(* IEC 61131-3 sources: OpenPLC_Sample_Programs/successed_ST (part 11) *)

        Pusher_states_t#Wait_Metal:
            Pusher2_transit := FALSE;
            Pusher_Timer3_IN := TRUE;
            Pusher_Timer3_PT := Pusher_Duration3;
            IF Pusher_Timer3_IN THEN
                Pusher_Timer3_Q := (Pusher_Timer3_ET = USINT#0);
                IF (Pusher_Timer3_ET > USINT#0) THEN
                    Pusher_Timer3_ET := (Pusher_Timer3_ET - USINT#1);
                ELSE
                    Pusher_Timer3_ET := USINT#0;
                END_IF;
            ELSE
                Pusher_Timer3_Q := FALSE;
                Pusher_Timer3_ET := Pusher_Timer3_PT;
            END_IF;
            Pusher_interconnect3 := Pusher_Timer3_Q;
            IF Pusher_interconnect3 THEN
                Pusher2_transit := TRUE;
                Pusher2_state := Pusher_states_t#Reset_interconnect_Slide3_Metal;
            END_IF;

        Pusher_states_t#Wait_White:
            Pusher2_transit := FALSE;
            Pusher_Timer3_IN := TRUE;
            Pusher_Timer3_PT := Pusher_Duration3;
            IF Pusher_Timer3_IN THEN
                Pusher_Timer3_Q := (Pusher_Timer3_ET = USINT#0);
                IF (Pusher_Timer3_ET > USINT#0) THEN
                    Pusher_Timer3_ET := (Pusher_Timer3_ET - USINT#1);
                ELSE
                    Pusher_Timer3_ET := USINT#0;
                END_IF;
            ELSE
                Pusher_Timer3_Q := FALSE;
                Pusher_Timer3_ET := Pusher_Timer3_PT;
            END_IF;
            Pusher_interconnect3 := Pusher_Timer3_Q;
            IF Pusher_interconnect3 THEN
                Pusher2_transit := TRUE;
                Pusher2_state := Pusher_states_t#Reset_interconnect_Slide3_White;
            END_IF;

        Pusher_states_t#Wait_Y1_Black:
            Pusher2_transit := FALSE;
            IF (Pusher_PusherY1 = TRUE) THEN
                Pusher_Timer3_IN := Pusher_PusherY1;
                Pusher_Timer3_PT := Pusher_Duration3;
                IF Pusher_Timer3_IN THEN
                    Pusher_Timer3_Q := (Pusher_Timer3_ET = USINT#0);
                    IF (Pusher_Timer3_ET > USINT#0) THEN
                        Pusher_Timer3_ET := (Pusher_Timer3_ET - USINT#1);
                    ELSE
                        Pusher_Timer3_ET := USINT#0;
                    END_IF;
                ELSE
                    Pusher_Timer3_Q := FALSE;
                    Pusher_Timer3_ET := Pusher_Timer3_PT;
                END_IF;
                Pusher_interconnect3 := Pusher_Timer3_Q;
            END_IF;
            IF Pusher_interconnect3 THEN
                Pusher2_transit := TRUE;
                Pusher2_state := Pusher_states_t#PusherY1_Move_In_Black;
            END_IF;

        Pusher_states_t#Wait_Y1_Metal:
            Pusher2_transit := FALSE;
            IF (Pusher_PusherY1 = TRUE) THEN
                Pusher_Timer3_IN := Pusher_PusherY1;
                Pusher_Timer3_PT := Pusher_Duration3;
                IF Pusher_Timer3_IN THEN
                    Pusher_Timer3_Q := (Pusher_Timer3_ET = USINT#0);
                    IF (Pusher_Timer3_ET > USINT#0) THEN
                        Pusher_Timer3_ET := (Pusher_Timer3_ET - USINT#1);
                    ELSE
                        Pusher_Timer3_ET := USINT#0;
                    END_IF;
                ELSE
                    Pusher_Timer3_Q := FALSE;
                    Pusher_Timer3_ET := Pusher_Timer3_PT;
                END_IF;
                Pusher_interconnect3 := Pusher_Timer3_Q;
            END_IF;
            IF Pusher_interconnect3 THEN
                Pusher2_transit := TRUE;
                Pusher2_state := Pusher_states_t#PusherY1_Move_In_Metal;
            END_IF;

        Pusher_states_t#Wait_Y1_White:
            Pusher2_transit := FALSE;
            IF (Pusher_PusherY1 = TRUE) THEN
                Pusher_Timer3_IN := Pusher_PusherY1;
                Pusher_Timer3_PT := Pusher_Duration3;
                IF Pusher_Timer3_IN THEN
                    Pusher_Timer3_Q := (Pusher_Timer3_ET = USINT#0);
                    IF (Pusher_Timer3_ET > USINT#0) THEN
                        Pusher_Timer3_ET := (Pusher_Timer3_ET - USINT#1);
                    ELSE
                        Pusher_Timer3_ET := USINT#0;
                    END_IF;
                ELSE
                    Pusher_Timer3_Q := FALSE;
                    Pusher_Timer3_ET := Pusher_Timer3_PT;
                END_IF;
                Pusher_interconnect3 := Pusher_Timer3_Q;
            END_IF;
            IF Pusher_interconnect3 THEN
                Pusher2_transit := TRUE;
                Pusher2_state := Pusher_states_t#PusherY1_Move_In_White;
            END_IF;

        Pusher_states_t#Wait_Y2_Black:
            Pusher2_transit := FALSE;
            IF (Pusher_PusherY2 = TRUE) THEN
                Pusher_Timer3_IN := Pusher_PusherY2;
                Pusher_Timer3_PT := Pusher_Duration3;
                IF Pusher_Timer3_IN THEN
                    Pusher_Timer3_Q := (Pusher_Timer3_ET = USINT#0);
                    IF (Pusher_Timer3_ET > USINT#0) THEN
                        Pusher_Timer3_ET := (Pusher_Timer3_ET - USINT#1);
                    ELSE
                        Pusher_Timer3_ET := USINT#0;
                    END_IF;
                ELSE
                    Pusher_Timer3_Q := FALSE;
                    Pusher_Timer3_ET := Pusher_Timer3_PT;
                END_IF;
                Pusher_interconnect3 := Pusher_Timer3_Q;
            END_IF;
            IF Pusher_interconnect3 THEN
                Pusher2_transit := TRUE;
                Pusher2_state := Pusher_states_t#PusherY2_Move_In_Black;
            END_IF;

        Pusher_states_t#Wait_Y2_Metal:
            Pusher2_transit := FALSE;
            IF (Pusher_PusherY2 = TRUE) THEN
                Pusher_Timer3_IN := Pusher_PusherY2;
                Pusher_Timer3_PT := Pusher_Duration3;
                IF Pusher_Timer3_IN THEN
                    Pusher_Timer3_Q := (Pusher_Timer3_ET = USINT#0);
                    IF (Pusher_Timer3_ET > USINT#0) THEN
                        Pusher_Timer3_ET := (Pusher_Timer3_ET - USINT#1);
                    ELSE
                        Pusher_Timer3_ET := USINT#0;
                    END_IF;
                ELSE
                    Pusher_Timer3_Q := FALSE;
                    Pusher_Timer3_ET := Pusher_Timer3_PT;
                END_IF;
                Pusher_interconnect3 := Pusher_Timer3_Q;
            END_IF;
            IF Pusher_interconnect3 THEN
                Pusher2_transit := TRUE;
                Pusher2_state := Pusher_states_t#PusherY2_Move_In_Metal;
            END_IF;

        Pusher_states_t#Wait_Y2_White:
            Pusher2_transit := FALSE;
            IF (Pusher_PusherY2 = TRUE) THEN
                Pusher_Timer3_IN := Pusher_PusherY2;
                Pusher_Timer3_PT := Pusher_Duration3;
                IF Pusher_Timer3_IN THEN
                    Pusher_Timer3_Q := (Pusher_Timer3_ET = USINT#0);
                    IF (Pusher_Timer3_ET > USINT#0) THEN
                        Pusher_Timer3_ET := (Pusher_Timer3_ET - USINT#1);
                    ELSE
                        Pusher_Timer3_ET := USINT#0;
                    END_IF;
                ELSE
                    Pusher_Timer3_Q := FALSE;
                    Pusher_Timer3_ET := Pusher_Timer3_PT;
                END_IF;
                Pusher_interconnect3 := Pusher_Timer3_Q;
            END_IF;
            IF Pusher_interconnect3 THEN
                Pusher2_transit := TRUE;
                Pusher2_state := Pusher_states_t#PusherY2_Move_In_White;
            END_IF;

            END_CASE;
    IF ((Actuator_SorterGreenLampConveyor AND Actuator_MagazinGreenLamp) AND Actuator_StampGreenLamp) THEN
        IF (((Stamp_StartCommandStamp AND Crane_StartCommandCrane) AND Conveyor_StartCommandConveyor) AND Mag_StartCommandMagazin) THEN
            Crane_StartVar := TRUE;
            Conveyor_StartVar := TRUE;
            Mag_StartVar := TRUE;
            Pusher_StartVar := TRUE;
            Stamp_StartVar := TRUE;
            DIAGNOSIS_ACTIVE := TRUE;
        END_IF;
    END_IF;
    Crane_SFCReset := FALSE;
    Conveyor_SFCReset := FALSE;
    Mag_SFCReset := FALSE;
    Pusher_SFCReset := FALSE;
    Stamp_SFCReset := FALSE;

    Crane_AnalogCranePressure := PARAMETER_CRANE_PRESSURE_METALLIC;

ELSIF ((NOT Sensor_SorterEmergencyStop OR NOT Sensor_StampEmergencyStop) OR NOT Sensor_MagazinEmergencyStop) THEN
    Actuator_MagazinSlider := FALSE;
    Actuator_CraneLower := FALSE;
    Actuator_MagazinVacuumOn := FALSE;
    Actuator_MagazinVacuumOff := TRUE;
    Actuator_MagazinGreenLamp := FALSE;
    Actuator_CraneTurnCounterclockwise := FALSE;
    Actuator_CraneTurnClockwise := FALSE;
    Actuator_SorterConveyorTowardsStacker := FALSE;
    Actuator_SorterConveyorTowardsCrane := FALSE;
    Actuator_SorterGreenLampConveyor := FALSE;
    Actuator_PusherY1 := FALSE;
    Actuator_PusherY2 := FALSE;
    Actuator_StampSliderMovedOut := TRUE;
    Actuator_StampSliderMovedIn := FALSE;
    Actuator_StampGreenLamp := FALSE;
    Actuator_StampPusher := FALSE;
    Actuator_AnalogCranePressure := 0;
    Crane_SFCReset := TRUE;
    Conveyor_SFCReset := TRUE;
    Mag_SFCReset := TRUE;
    Pusher_SFCReset := TRUE;
    Stamp_SFCReset := TRUE;
    Crane_StartVar := FALSE;
    Conveyor_StartVar := FALSE;
    Mag_StartVar := FALSE;
    Pusher_StartVar := FALSE;
    Stamp_StartVar := FALSE;
END_IF;

END_PROGRAM

CONFIGURATION Config0
  RESOURCE Res0 ON PLC
    TASK task0(INTERVAL := T#50ms, PRIORITY := 0);
    PROGRAM instance0 WITH task0 : Main;
  END_RESOURCE
END_CONFIGURATION

(* ---- Code_3.st ---- *)
TYPE
Crane3_states_t : (Crane_Init,Crane_Go_Up , Crane_Init_2 , Crane_Lift_At_Stamp
, Crane_Lift_Conveyor , Crane_Lift_Magazin , Crane_Lift_Magazin_Metallic ,
Crane_Lower , Crane_On_Conveyor , Crane_On_Conveyor_Metallic ,
Crane_On_Stamp_Metallic , Crane_Turn_Left_From_Stamp , Crane_Turn_Left_Metallic
, Crane_Turn_Left_NOT_Metallic , Init , Interstep , Interstep_2 ,
Interstep_Check_Workpiece , Lower_Crane , Reset_interconnect , Start_Crane ,
Step0 , Step2 , Suck_At_Stamp , TimeDelay , Turn_Right , Wait_At_Stamp , pause ,
release , release_Workpiece);
END_TYPE

PROGRAM Crane3
    VAR  Duration1 : TIME := T#1s500ms; END_VAR
    VAR  SFCInit : BOOL; END_VAR
    VAR  TimeDelay_Timer : TON; END_VAR
    VAR  TimeDelay_Timer_Duration : TIME := T#50ms; END_VAR
    VAR  TimeDelay_Timer_interconnect : BOOL; END_VAR
    VAR  Timer1 : TON; END_VAR
    VAR  _state : Crane3_states_t; END_VAR
    VAR  _transit : BOOL; END_VAR
    VAR  actualtime1 : TIME; END_VAR
    VAR  interconnect : BOOL; END_VAR
    VAR  interconnectCraneStartCommand : BOOL; END_VAR

    VAR_INPUT  CraneDown : BOOL; END_VAR
    VAR_INPUT  CraneOnConveyor : BOOL; END_VAR
    VAR_INPUT  CraneOnMagazin : BOOL; END_VAR
    VAR_INPUT  CranePositionStamp : BOOL; END_VAR
    VAR_INPUT  CraneSucked : BOOL; END_VAR
    VAR_INPUT  CraneUp : BOOL; END_VAR
    VAR_INPUT  MagazinCapacitiveSensor : BOOL; END_VAR
    VAR_INPUT  SFCReset : BOOL; END_VAR
    VAR_INPUT  SliderMovedOut : BOOL; END_VAR
    VAR_INPUT  SliderNotMovedOut : BOOL; END_VAR
    VAR_INPUT  StampLowered : BOOL; END_VAR
    VAR_INPUT  StampSliderFilled : BOOL; END_VAR
    VAR_INPUT  StartButtonMagazin : BOOL; END_VAR
    VAR_INPUT  StartVar : BOOL; END_VAR
    VAR_INPUT  WorkpieceReady : BOOL; END_VAR

    VAR_OUTPUT  CraneLower : BOOL; END_VAR
    VAR_OUTPUT  CraneTurnClockwise : BOOL; END_VAR
    VAR_OUTPUT  CraneTurnCounterclockwise : BOOL; END_VAR
    VAR_OUTPUT  MagazinVacuumOff : BOOL; END_VAR
    VAR_OUTPUT  MagazinVacuumOn : BOOL; END_VAR
    VAR_OUTPUT  StartCommandCrane : BOOL; END_VAR

    CASE _state OF
        Crane3_states_t#Crane_Go_Up:
            _transit := FALSE;
            CraneLower := FALSE;
            IF CraneUp THEN
                _transit := TRUE;
                _state := Crane3_states_t#pause;
            END_IF;
        Crane3_states_t#Crane_Init:
            _transit := FALSE;
            CraneLower := TRUE;
            interconnectCraneStartCommand := FALSE;
            IF CraneDown THEN
                _transit := TRUE;
                _state := Crane3_states_t#Crane_Init_2;
            END_IF;
        Crane3_states_t#Crane_Init_2:
            _transit := FALSE;
            CraneLower := FALSE;
            IF CraneUp THEN
                _transit := TRUE;
                _state := Crane3_states_t#Interstep;
            END_IF;
        Crane3_states_t#Crane_Lift_At_Stamp:
            _transit := FALSE;
            CraneLower := FALSE;
            IF CraneUp THEN
                _transit := TRUE;
                _state := Crane3_states_t#Crane_Turn_Left_From_Stamp;
            END_IF;
        Crane3_states_t#Crane_Lift_Conveyor:
            _transit := FALSE;
            CraneLower := FALSE;
            IF TRUE THEN
                _transit := TRUE;
                _state := Crane3_states_t#Interstep;
            END_IF;
        Crane3_states_t#Crane_Lift_Magazin:
            _transit := FALSE;
            CraneLower := FALSE;
            IF CraneUp THEN
                _transit := TRUE;
                _state := Crane3_states_t#Crane_Turn_Left_NOT_Metallic;
            END_IF;
        Crane3_states_t#Crane_Lift_Magazin_Metallic:
            _transit := FALSE;
            CraneLower := FALSE;
            IF CraneUp THEN
                _transit := TRUE;
                _state := Crane3_states_t#Crane_Turn_Left_Metallic;
            END_IF;
        Crane3_states_t#Crane_Lower:
            _transit := FALSE;
            MagazinVacuumOn := TRUE;
            MagazinVacuumOff := FALSE;
            CraneLower := TRUE;
            IF CraneSucked THEN
                _transit := TRUE;
                _state := Crane3_states_t#Step0;
            END_IF;
        Crane3_states_t#Crane_On_Conveyor:
            _transit := FALSE;
            CraneTurnCounterclockwise := FALSE;
            CraneTurnClockwise := FALSE;
            CraneLower := TRUE;
            IF CraneDown THEN
                _transit := TRUE;
                _state := Crane3_states_t#release;
            END_IF;
        Crane3_states_t#Crane_On_Conveyor_Metallic:
            _transit := FALSE;
            CraneTurnCounterclockwise := FALSE;
            CraneTurnClockwise := FALSE;
            CraneLower := TRUE;
            IF CraneDown THEN
                _transit := TRUE;
                _state := Crane3_states_t#release;
            END_IF;
        Crane3_states_t#Crane_On_Stamp_Metallic:
            _transit := FALSE;
            CraneTurnCounterclockwise := FALSE;
            CraneTurnClockwise := FALSE;
            CraneLower := TRUE;
            IF CraneDown THEN
                _transit := TRUE;
                _state := Crane3_states_t#release_Workpiece;
            END_IF;
        Crane3_states_t#Crane_Turn_Left_From_Stamp:
            _transit := FALSE;
            CraneTurnClockwise := TRUE;
            CraneTurnCounterclockwise := FALSE;
            IF CraneOnConveyor THEN
                _transit := TRUE;
                _state := Crane3_states_t#Crane_On_Conveyor_Metallic;
            END_IF;
        Crane3_states_t#Crane_Turn_Left_Metallic:
            _transit := FALSE;
            CraneTurnCounterclockwise := TRUE;
            CraneTurnClockwise := FALSE;
            IF CranePositionStamp THEN
                _transit := TRUE;
                _state := Crane3_states_t#Crane_On_Stamp_Metallic;
            END_IF;
        Crane3_states_t#Crane_Turn_Left_NOT_Metallic:
            _transit := FALSE;
            CraneTurnCounterclockwise := TRUE;
            CraneTurnClockwise := FALSE;
            IF CraneOnConveyor THEN
                _transit := TRUE;
                _state := Crane3_states_t#Crane_On_Conveyor;
            END_IF;
        Crane3_states_t#Init:
            _transit := FALSE;
            IF TRUE THEN
                _transit := TRUE;
                _state := Crane3_states_t#Start_Crane;
            END_IF;
        Crane3_states_t#Interstep:
            _transit := FALSE;
            StartCommandCrane := TRUE;
            IF StartVar THEN
                _transit := TRUE;
                _state := Crane3_states_t#Interstep_2;
            END_IF;
        Crane3_states_t#Interstep_2:
            _transit := FALSE;
            IF SliderMovedOut THEN
                _transit := TRUE;
                _state := Crane3_states_t#TimeDelay;
            END_IF;
        Crane3_states_t#Interstep_Check_Workpiece:
            _transit := FALSE;
            CraneTurnClockwise := FALSE;
            CraneTurnCounterclockwise := FALSE;
            IF (NOT WorkpieceReady AND StampSliderFilled) THEN
                _transit := TRUE;
                _state := Crane3_states_t#Wait_At_Stamp;
            ELSIF (NOT WorkpieceReady AND NOT StampSliderFilled) THEN
                _transit := TRUE;
                _state := Crane3_states_t#Step2;
            ELSIF WorkpieceReady THEN
                _transit := TRUE;
                _state := Crane3_states_t#Crane_Lower;
            END_IF;
        Crane3_states_t#Lower_Crane:
            _transit := FALSE;
            CraneLower := TRUE;
            IF CraneDown THEN
                _transit := TRUE;
                _state := Crane3_states_t#Suck_At_Stamp;
            END_IF;
        Crane3_states_t#Reset_interconnect:
            _transit := FALSE;
            interconnect := FALSE;
            Timer1(IN := FALSE, PT := TIME#1ms);
            IF SliderMovedOut THEN
                _transit := TRUE;
                _state := Crane3_states_t#Lower_Crane;
            END_IF;
        Crane3_states_t#Start_Crane:
            _transit := FALSE;
            CraneLower := FALSE;
            MagazinVacuumOff := TRUE;
            MagazinVacuumOn := FALSE;
            CraneTurnCounterclockwise := FALSE;
            CraneTurnClockwise := FALSE;
            StartVar := FALSE;
            StartCommandCrane := FALSE;
            IF (StartButtonMagazin = TRUE) THEN
                interconnectCraneStartCommand := TRUE;
            END_IF;
            IF interconnectCraneStartCommand THEN
                _transit := TRUE;
                _state := Crane3_states_t#Crane_Init;
            END_IF;
        Crane3_states_t#Step0:
            _transit := FALSE;
            IF NOT MagazinCapacitiveSensor THEN
                _transit := TRUE;
                _state := Crane3_states_t#Crane_Lift_Magazin;
            ELSIF MagazinCapacitiveSensor THEN
                _transit := TRUE;
                _state := Crane3_states_t#Crane_Lift_Magazin_Metallic;
            END_IF;
        Crane3_states_t#Step2:
            _transit := FALSE;
            IF TRUE THEN
                _transit := TRUE;
                _state := Crane3_states_t#Start_Crane;
            END_IF;
        Crane3_states_t#Suck_At_Stamp:
            _transit := FALSE;
            MagazinVacuumOn := TRUE;
            MagazinVacuumOff := FALSE;
            IF CraneSucked THEN
                _transit := TRUE;
                _state := Crane3_states_t#Crane_Lift_At_Stamp;
            END_IF;
        Crane3_states_t#TimeDelay:
            _transit := FALSE;
            TimeDelay_Timer(IN := TRUE, PT := TimeDelay_Timer_Duration);
            TimeDelay_Timer_interconnect := TimeDelay_Timer.Q;
            IF TimeDelay_Timer_interconnect THEN
                _transit := TRUE;
                _state := Crane3_states_t#Turn_Right;
            END_IF;
        Crane3_states_t#Turn_Right:
             _transit := FALSE;
             CraneTurnClockwise := TRUE;
             CraneTurnCounterclockwise := FALSE;
             IF CraneOnMagazin THEN
                _transit := TRUE;
                _state := Crane3_states_t#Interstep_Check_Workpiece;
             END_IF;
        Crane3_states_t#Wait_At_Stamp:
            _transit := FALSE;
            IF TRUE THEN
                _transit := TRUE;
                _state := Crane3_states_t#pause;
            END_IF;
        Crane3_states_t#pause:
            _transit := FALSE;
            Timer1(IN := CraneUp, PT := Duration1);
            interconnect := Timer1.Q;
            IF interconnect THEN
                _transit := TRUE;
                _state := Crane3_states_t#Reset_interconnect;
            END_IF;
        Crane3_states_t#release:
            _transit := FALSE;
            MagazinVacuumOff := TRUE;
            MagazinVacuumOn := FALSE;
            IF TRUE THEN
                _transit := TRUE;
                _state := Crane3_states_t#Crane_Lift_Conveyor;
            END_IF;
        Crane3_states_t#release_Workpiece:
            _transit := FALSE;
            MagazinVacuumOff := TRUE;
            MagazinVacuumOn := FALSE;
            IF TRUE THEN
                _transit := TRUE;
                _state := Crane3_states_t#Crane_Go_Up;
            END_IF;
        END_CASE;
END_PROGRAM

CONFIGURATION Config0
  RESOURCE Res0 ON PLC
    TASK task0(INTERVAL := T#50ms, PRIORITY := 0);
    PROGRAM instance0 WITH task0 : Crane3;
  END_RESOURCE
END_CONFIGURATION

(* ---- Code_5.st ---- *)
TYPE
Crane5_states_t : (Crane_Init ,Crane_Go_Up ,  Crane_Init_2 , Crane_Lift_At_Stamp
, Crane_Lift_Conveyor , Crane_Lift_Conveyor_Black , Crane_Lift_Magazin ,
Crane_Lift_Magazin_Metallic , Crane_Lift_NOT_Metallic_Black , Crane_Lower ,
Crane_On_Conveyor , Crane_On_Conveyor_Metallic ,
Crane_On_Conveyor_Not_Metallica_Black , Crane_On_Stamp_Metallic ,
Crane_On_Stamp_Stop_Black , Crane_Turn_Left_Back_To_Stamp ,
Crane_Turn_Left_From_Stamp , Crane_Turn_Left_Metallic ,
Crane_Turn_Left_NOT_Metallic , Crane_Turn_Left_NOT_Metallic_Black , Init ,
Interstep , Interstep_2 , Last_Workpiece_At_Stamp , Lower_Crane , Magazin_Stop ,
Magazin_Stop_Black , No_Workpiece_ready , Reset_interconnect , Start_Crane ,
Step0 , Suck_At_Stamp , TimeDelay , Turn_Right , Turn_Right_Black , pause ,
release , release_Black , release_Workpiece);
END_TYPE

PROGRAM Crane5
    VAR  CranTurnClockwise : BOOL; END_VAR
    VAR_INPUT  CraneDown : BOOL; END_VAR
    VAR_OUTPUT  CraneLower : BOOL; END_VAR
    VAR_INPUT  CraneOnConveyor : BOOL; END_VAR
    VAR_INPUT  CraneOnMagazin : BOOL; END_VAR
    VAR_INPUT  CranePositionStamp : BOOL; END_VAR
    VAR_INPUT  CraneSucked : BOOL; END_VAR
    VAR_OUTPUT  CraneTurnClockwise : BOOL; END_VAR
    VAR_OUTPUT  CraneTurnCounterclockwise : BOOL; END_VAR
    VAR_INPUT  CraneUp : BOOL; END_VAR
    VAR  Duration1 : TIME := TIME#1s500ms; END_VAR
    VAR_INPUT  MagazinCapacitiveSensor : BOOL; END_VAR
    VAR_OUTPUT  MagazinVacuumOff : BOOL; END_VAR
    VAR_OUTPUT  MagazinVacuumOn : BOOL; END_VAR
    VAR  SFCInit : BOOL; END_VAR
    VAR_INPUT  SFCReset : BOOL; END_VAR
    VAR_INPUT  SliderMovedOut : BOOL; END_VAR
    VAR_INPUT  SliderNotMovedOut : BOOL; END_VAR
    VAR_INPUT  StampLowered : BOOL; END_VAR
    VAR_INPUT  StampSliderFilled : BOOL; END_VAR
    VAR_INPUT  StartButtonMagazin : BOOL; END_VAR
    VAR_OUTPUT  StartCommandCrane : BOOL; END_VAR
    VAR_INPUT  StartVar : BOOL; END_VAR
    VAR  TimeDelay_Timer : TON; END_VAR
    VAR  TimeDelay_Timer_Duration : TIME := TIME#50.0ms; END_VAR
    VAR  TimeDelay_Timer_interconnect : BOOL; END_VAR
    VAR  Timer1 : TON; END_VAR
    VAR_INPUT  WorkpieceReady : BOOL; END_VAR
    VAR  _state : Crane5_states_t; END_VAR
    VAR  _transit : BOOL; END_VAR
    VAR  actualtime1 : TIME; END_VAR
    VAR  interconnect : BOOL; END_VAR
    VAR  interconnectCraneStartCommand : BOOL; END_VAR

    CASE _state OF
        Crane5_states_t#Crane_Go_Up:
            _transit := FALSE;
            CraneLower := FALSE;
            IF (CraneUp AND (MagazinCapacitiveSensor OR NOT WorkpieceReady)) THEN
                _transit := TRUE;
                _state := Crane5_states_t#pause;
            ELSIF ((CraneUp AND NOT MagazinCapacitiveSensor) AND WorkpieceReady) THEN
                _transit := TRUE;
                _state := Crane5_states_t#Turn_Right_Black;
            END_IF;
        Crane5_states_t#Crane_Init:
            _transit := FALSE;
            CraneLower := TRUE;
            interconnectCraneStartCommand := FALSE;
            IF CraneDown THEN
                _transit := TRUE;
                _state := Crane5_states_t#Crane_Init_2;
            END_IF;
        Crane5_states_t#Crane_Init_2:
            _transit := FALSE;
            CraneLower := FALSE;
            IF CraneUp THEN
                _transit := TRUE;
                _state := Crane5_states_t#Interstep;
            END_IF;
        Crane5_states_t#Crane_Lift_At_Stamp:
            _transit := FALSE;
            CraneLower := FALSE;
            IF CraneUp THEN
                _transit := TRUE;
                _state := Crane5_states_t#Crane_Turn_Left_From_Stamp;
            END_IF;
        Crane5_states_t#Crane_Lift_Conveyor:
            _transit := FALSE;
            CraneLower := FALSE;
            IF TRUE THEN
                _transit := TRUE;
                _state := Crane5_states_t#Interstep;
            END_IF;
        Crane5_states_t#Crane_Lift_Conveyor_Black:
            _transit := FALSE;
            CraneLower := FALSE;
            IF CraneUp THEN
                _transit := TRUE;
                _state := Crane5_states_t#Crane_Turn_Left_Back_To_Stamp;
            END_IF;
        Crane5_states_t#Crane_Lift_Magazin:
            _transit := FALSE;
            CraneLower := FALSE;
            IF CraneUp THEN
                _transit := TRUE;
                _state := Crane5_states_t#Crane_Turn_Left_NOT_Metallic;
            END_IF;
        Crane5_states_t#Crane_Lift_Magazin_Metallic:
            _transit := FALSE;
            CraneLower := FALSE;
            IF CraneUp THEN
                _transit := TRUE;
                _state := Crane5_states_t#Crane_Turn_Left_Metallic;
            END_IF;
        Crane5_states_t#Crane_Lift_NOT_Metallic_Black:
            _transit := FALSE;
            CraneLower := FALSE;
            IF CraneUp THEN
                _transit := TRUE;
                _state := Crane5_states_t#Crane_Turn_Left_NOT_Metallic_Black;
            END_IF;
        Crane5_states_t#Crane_Lower:
            _transit := FALSE;
            MagazinVacuumOn := TRUE;
            MagazinVacuumOff := FALSE;
            CraneLower := TRUE;
            IF CraneSucked THEN
                _transit := TRUE;
                _state := Crane5_states_t#Step0;
            END_IF;
        Crane5_states_t#Crane_On_Conveyor:
            _transit := FALSE;
            CraneTurnCounterclockwise := FALSE;
            CraneTurnClockwise := FALSE;
            CraneLower := TRUE;
            IF CraneDown THEN
                _transit := TRUE;
                _state := Crane5_states_t#release;
            END_IF;
        Crane5_states_t#Crane_On_Conveyor_Metallic:
            _transit := FALSE;
            CraneTurnCounterclockwise := FALSE;
            CraneTurnClockwise := FALSE;
            CraneLower := TRUE;
            IF CraneDown THEN
                _transit := TRUE;
                _state := Crane5_states_t#release;
            END_IF;
        Crane5_states_t#Crane_On_Conveyor_Not_Metallica_Black:
            _transit := FALSE;
            CraneTurnCounterclockwise := FALSE;
            CraneTurnClockwise := FALSE;
            CraneLower := TRUE;
            IF CraneDown THEN
                _transit := TRUE;
                _state := Crane5_states_t#release_Black;
            END_IF;
        Crane5_states_t#Crane_On_Stamp_Metallic:
            _transit := FALSE;
            CraneTurnCounterclockwise := FALSE;
            CraneTurnClockwise := FALSE;
            CraneLower := TRUE;
            IF CraneDown THEN
                _transit := TRUE;
                _state := Crane5_states_t#release_Workpiece;
            END_IF;
        Crane5_states_t#Crane_On_Stamp_Stop_Black:
            _transit := FALSE;
            CraneTurnClockwise := FALSE;
            CraneTurnCounterclockwise := FALSE;
            IF TRUE THEN
                _transit := TRUE;
                _state := Crane5_states_t#Reset_interconnect;
            END_IF;
        Crane5_states_t#Crane_Turn_Left_Back_To_Stamp:
            _transit := FALSE;
            CraneTurnCounterclockwise := TRUE;
            CraneTurnClockwise := FALSE;
            IF CranePositionStamp THEN
                _transit := TRUE;
                _state := Crane5_states_t#Crane_On_Stamp_Stop_Black;
            END_IF;
        Crane5_states_t#Crane_Turn_Left_From_Stamp:
            _transit := FALSE;
            CraneTurnClockwise := TRUE;
            CraneTurnCounterclockwise := FALSE;
            IF CraneOnConveyor THEN
                _transit := TRUE;
                _state := Crane5_states_t#Crane_On_Conveyor_Metallic;
            END_IF;
        Crane5_states_t#Crane_Turn_Left_Metallic:
            _transit := FALSE;
            CraneTurnCounterclockwise := TRUE;
            CraneTurnClockwise := FALSE;
            IF CranePositionStamp THEN
                _transit := TRUE;
                _state := Crane5_states_t#Crane_On_Stamp_Metallic;
            END_IF;
        Crane5_states_t#Crane_Turn_Left_NOT_Metallic:
            _transit := FALSE;
            CraneTurnCounterclockwise := TRUE;
            CraneTurnClockwise := FALSE;
            IF CraneOnConveyor THEN
                _transit := TRUE;
                _state := Crane5_states_t#Crane_On_Conveyor;
            END_IF;
        Crane5_states_t#Crane_Turn_Left_NOT_Metallic_Black:
            _transit := FALSE;
            CraneTurnCounterclockwise := TRUE;
            CraneTurnClockwise := FALSE;
            IF CraneOnConveyor THEN
                _transit := TRUE;
                _state := Crane5_states_t#Crane_On_Conveyor_Not_Metallica_Black;
            END_IF;
        Crane5_states_t#Init:
            _transit := FALSE;
            IF TRUE THEN
                _transit := TRUE;
                _state := Crane5_states_t#Start_Crane;
            END_IF;
        Crane5_states_t#Interstep:
            _transit := FALSE;
            StartCommandCrane := TRUE;
            IF StartVar THEN
                _transit := TRUE;
                _state := Crane5_states_t#Interstep_2;
            END_IF;
        Crane5_states_t#Interstep_2:
            _transit := FALSE;
            IF SliderMovedOut THEN
                _transit := TRUE;
                _state := Crane5_states_t#TimeDelay;
            END_IF;
        Crane5_states_t#Last_Workpiece_At_Stamp:
            _transit := FALSE;
            IF TRUE THEN
                _transit := TRUE;
                _state := Crane5_states_t#pause;
            END_IF;
        Crane5_states_t#Lower_Crane:
            _transit := FALSE;
            CraneLower := TRUE;
            IF CraneDown THEN
                _transit := TRUE;
                _state := Crane5_states_t#Suck_At_Stamp;
            END_IF;
        Crane5_states_t#Magazin_Stop:
            _transit := FALSE;
            CraneTurnClockwise := FALSE;
            CraneTurnCounterclockwise := FALSE;
            IF WorkpieceReady THEN
                _transit := TRUE;
                _state := Crane5_states_t#Crane_Lower;
            ELSIF (NOT WorkpieceReady AND NOT StampSliderFilled) THEN
                _transit := TRUE;
                _state := Crane5_states_t#No_Workpiece_ready;
            ELSIF (NOT WorkpieceReady AND StampSliderFilled) THEN
                _transit := TRUE;
                _state := Crane5_states_t#Last_Workpiece_At_Stamp;
            END_IF;
        Crane5_states_t#Magazin_Stop_Black:
            _transit := FALSE;
            CraneTurnClockwise := FALSE;
            CraneTurnCounterclockwise := FALSE;
            MagazinVacuumOn := TRUE;
            MagazinVacuumOff := FALSE;
            CraneLower := TRUE;
            IF CraneSucked THEN
                _transit := TRUE;
                _state := Crane5_states_t#Crane_Lift_NOT_Metallic_Black;
            END_IF;
        Crane5_states_t#No_Workpiece_ready:
            _transit := FALSE;
            IF TRUE THEN
                _transit := TRUE;
                _state := Crane5_states_t#Start_Crane;
            END_IF;
        Crane5_states_t#Reset_interconnect:
            _transit := FALSE;
            interconnect := FALSE;
            Timer1(IN := FALSE, PT := TIME#1.0ms);
            IF SliderMovedOut THEN
                _transit := TRUE;
                _state := Crane5_states_t#Lower_Crane;
            END_IF;
        Crane5_states_t#Start_Crane:
            _transit := FALSE;
            CraneLower := FALSE;
            MagazinVacuumOff := TRUE;
            MagazinVacuumOn := FALSE;
            CraneTurnCounterclockwise := FALSE;
            CraneTurnClockwise := FALSE;
            StartVar := FALSE;
            StartCommandCrane := FALSE;
            IF (StartButtonMagazin = TRUE) THEN
                interconnectCraneStartCommand := TRUE;
            END_IF;
            IF interconnectCraneStartCommand THEN
                _transit := TRUE;
                _state := Crane5_states_t#Crane_Init;
            END_IF;
        Crane5_states_t#Step0:
            _transit := FALSE;
            IF NOT MagazinCapacitiveSensor THEN
                _transit := TRUE;
                _state := Crane5_states_t#Crane_Lift_Magazin;
            ELSIF MagazinCapacitiveSensor THEN
                _transit := TRUE;
                _state := Crane5_states_t#Crane_Lift_Magazin_Metallic;
            END_IF;
        Crane5_states_t#Suck_At_Stamp:
            _transit := FALSE;
            MagazinVacuumOn := TRUE;
            MagazinVacuumOff := FALSE;
            IF CraneSucked THEN
                _transit := TRUE;
                _state := Crane5_states_t#Crane_Lift_At_Stamp;
            END_IF;
        Crane5_states_t#TimeDelay:
            _transit := FALSE;
            TimeDelay_Timer(IN := TRUE, PT := TimeDelay_Timer_Duration);
            TimeDelay_Timer_interconnect := TimeDelay_Timer.Q;
            IF TimeDelay_Timer_interconnect THEN
                _transit := TRUE;
                _state := Crane5_states_t#Turn_Right;
            END_IF;
        Crane5_states_t#Turn_Right:
            _transit := FALSE;
            CraneTurnClockwise := TRUE;
            CraneTurnCounterclockwise := FALSE;
            IF CraneOnMagazin THEN
                _transit := TRUE;
                _state := Crane5_states_t#Magazin_Stop;
            END_IF;
        Crane5_states_t#Turn_Right_Black:
            _transit := FALSE;
            CraneTurnClockwise := TRUE;
            CraneTurnCounterclockwise := FALSE;
            IF CraneOnMagazin THEN
                _transit := TRUE;
                _state := Crane5_states_t#Magazin_Stop_Black;
            END_IF;
        Crane5_states_t#pause:
            _transit := FALSE;
            Timer1(IN := CraneUp, PT := Duration1);
            interconnect := Timer1.Q;
            IF interconnect THEN
                _transit := TRUE;
                _state := Crane5_states_t#Reset_interconnect;
            END_IF;
        Crane5_states_t#release:
            _transit := FALSE;
            MagazinVacuumOff := TRUE;
            MagazinVacuumOn := FALSE;
            IF TRUE THEN
                _transit := TRUE;
                _state := Crane5_states_t#Crane_Lift_Conveyor;
            END_IF;
        Crane5_states_t#release_Black:
            _transit := FALSE;
            MagazinVacuumOn := FALSE;
            MagazinVacuumOff := TRUE;
            IF TRUE THEN
                _transit := TRUE;
                _state := Crane5_states_t#Crane_Lift_Conveyor_Black;
            END_IF;
        Crane5_states_t#release_Workpiece:
            _transit := FALSE;
            MagazinVacuumOff := TRUE;
            MagazinVacuumOn := FALSE;
            IF TRUE THEN
                _transit := TRUE;
                _state := Crane5_states_t#Crane_Go_Up;
            END_IF;
    END_CASE;
END_PROGRAM

CONFIGURATION Config0
  RESOURCE Res0 ON PLC
    TASK task0(INTERVAL := T#50ms, PRIORITY := 0);
    PROGRAM instance0 WITH task0 : Crane5;
  END_RESOURCE
END_CONFIGURATION

(* ---- constantprogram.st ---- *)
PROGRAM CONSTANTPROGRAM
    VAR_INPUT
        I : INT;
    END_VAR

    VAR_OUTPUT
        O : INT;
        C : INT;
    END_VAR

    O := I;
    C := 42;

END_PROGRAM

CONFIGURATION Config0
  RESOURCE Res0 ON PLC
    TASK TASK0(INTERVAL := T#50MS, PRIORITY := 0);
    PROGRAM INSTANCE0 WITH TASK0 : CONSTANTPROGRAM;
  END_RESOURCE
END_CONFIGURATION

(* ---- Crane.st ---- *)
TYPE
    CRANE_STATES_T : (CRANE_GO_UP , CRANE_INIT , CRANE_INIT_2 , CRANE_LIFT_AT_STAMP , CRANE_LIFT_CONVEYOR , CRANE_LIFT_CONVEYOR_BLACK , CRANE_LIFT_MAGAZIN , CRANE_LIFT_MAGAZIN_METALLIC , CRANE_LIFT_NOT_METALLIC_BLACK , CRANE_LOWER , CRANE_ON_CONVEYOR , CRANE_ON_CONVEYOR_METALLIC , CRANE_ON_CONVEYOR_NOT_METALLICA_BLACK , CRANE_ON_STAMP_METALLIC , CRANE_ON_STAMP_STOP_BLACK , CRANE_TURN_LEFT_BACK_TO_STAMP , CRANE_TURN_LEFT_FROM_STAMP , CRANE_TURN_LEFT_METALLIC , CRANE_TURN_LEFT_NOT_METALLIC , CRANE_TURN_LEFT_NOT_METALLIC_BLACK , INIT , INTERSTEP , INTERSTEP_2 , LAST_WORKPIECE_AT_STAMP , LOWER_CRANE , MAGAZIN_STOP , MAGAZIN_STOP_BLACK , NO_WORKPIECE_READY , RESET_INTERCONNECT , START_CRANE , STEP0 , SUCK_AT_STAMP , TIMEDELAY , TURN_RIGHT , TURN_RIGHT_BLACK , PAUSE , RELEASE , RELEASE_BLACK , RELEASE_WORKPIECE);
END_TYPE

PROGRAM CRANE
    VAR  CRANTURNCLOCKWISE : BOOL; END_VAR
    VAR_INPUT  CRANEDOWN : BOOL; END_VAR
    VAR_OUTPUT  CRANELOWER : BOOL; END_VAR
    VAR_INPUT  CRANEONCONVEYOR : BOOL; END_VAR
    VAR_INPUT  CRANEONMAGAZIN : BOOL; END_VAR
    VAR_INPUT  CRANEPOSITIONSTAMP : BOOL; END_VAR
    VAR_INPUT  CRANESUCKED : BOOL; END_VAR
    VAR_OUTPUT  CRANETURNCLOCKWISE : BOOL; END_VAR
    VAR_OUTPUT  CRANETURNCOUNTERCLOCKWISE : BOOL; END_VAR
    VAR_INPUT  CRANEUP : BOOL; END_VAR
    VAR  DURATION1 : TIME := TIME#1S500MS; END_VAR
    VAR_INPUT  MAGAZINCAPACITIVESENSOR : BOOL; END_VAR
    VAR_OUTPUT  MAGAZINSLIDER : BOOL; END_VAR
    VAR_OUTPUT  MAGAZINVACUUMOFF : BOOL; END_VAR
    VAR_OUTPUT  MAGAZINVACUUMON : BOOL; END_VAR
    VAR  SFCINIT : BOOL; END_VAR
    VAR_INPUT  SFCRESET : BOOL; END_VAR
    VAR_INPUT  SLIDERMOVEDOUT : BOOL; END_VAR
    VAR_INPUT  SLIDERNOTMOVEDOUT : BOOL; END_VAR
    VAR_INPUT  STAMPLOWERED : BOOL; END_VAR
    VAR_INPUT  STAMPSLIDERFILLED : BOOL; END_VAR
    VAR_INPUT  STARTBUTTONMAGAZIN : BOOL; END_VAR
    VAR_OUTPUT  STARTCOMMANDCRANE : BOOL; END_VAR
    VAR_INPUT  STARTVAR : BOOL; END_VAR
    VAR  TIMEDELAY_TIMER : TON; END_VAR
    VAR  TIMEDELAY_TIMER_DURATION : TIME := TIME#50MS; END_VAR
    VAR  TIMEDELAY_TIMER_INTERCONNECT : BOOL; END_VAR
    VAR  TIMER1 : TON; END_VAR
    VAR_INPUT  WORKPIECEREADY : BOOL; END_VAR
    VAR  _STATE : CRANE_STATES_T := CRANE_STATES_T#INIT; END_VAR
    VAR  _TRANSIT : BOOL; END_VAR
    VAR  ACTUALTIME1 : TIME; END_VAR
    VAR  INTERCONNECT : BOOL; END_VAR
    VAR  INTERCONNECTCRANESTARTCOMMAND : BOOL; END_VAR

    IF SFCRESET THEN
        _STATE := CRANE_STATES_T#INIT;
    END_IF;

    CASE _STATE OF
        CRANE_STATES_T#CRANE_GO_UP:
            _TRANSIT := FALSE;
            CRANELOWER := FALSE;
            IF (CRANEUP AND (MAGAZINCAPACITIVESENSOR OR NOT WORKPIECEREADY)) THEN
                _TRANSIT := TRUE;
                _STATE := CRANE_STATES_T#PAUSE;
            ELSIF ((CRANEUP AND NOT MAGAZINCAPACITIVESENSOR) AND WORKPIECEREADY) THEN
                _TRANSIT := TRUE;
                _STATE := CRANE_STATES_T#TURN_RIGHT_BLACK;
            END_IF;

        CRANE_STATES_T#CRANE_INIT:
            _TRANSIT := FALSE;
            CRANELOWER := TRUE;
            INTERCONNECTCRANESTARTCOMMAND := FALSE;
            IF CRANEDOWN THEN
                _TRANSIT := TRUE;
                _STATE := CRANE_STATES_T#CRANE_INIT_2;
            END_IF;

        CRANE_STATES_T#CRANE_INIT_2:
            _TRANSIT := FALSE;
            CRANELOWER := FALSE;
            IF CRANEUP THEN
                _TRANSIT := TRUE;
                _STATE := CRANE_STATES_T#INTERSTEP;
            END_IF;

        CRANE_STATES_T#CRANE_LIFT_AT_STAMP:
            _TRANSIT := FALSE;
            CRANELOWER := FALSE;
            IF CRANEUP THEN
                _TRANSIT := TRUE;
                _STATE := CRANE_STATES_T#CRANE_TURN_LEFT_FROM_STAMP;
            END_IF;

        CRANE_STATES_T#CRANE_LIFT_CONVEYOR:
            _TRANSIT := FALSE;
            CRANELOWER := FALSE;
            IF TRUE THEN
                _TRANSIT := TRUE;
                _STATE := CRANE_STATES_T#INTERSTEP;
            END_IF;

        CRANE_STATES_T#CRANE_LIFT_CONVEYOR_BLACK:
            _TRANSIT := FALSE;
            CRANELOWER := FALSE;
            IF CRANEUP THEN
                _TRANSIT := TRUE;
                _STATE := CRANE_STATES_T#CRANE_TURN_LEFT_BACK_TO_STAMP;
            END_IF;

        CRANE_STATES_T#CRANE_LIFT_MAGAZIN:
            _TRANSIT := FALSE;
            CRANELOWER := FALSE;
            IF CRANEUP THEN
                _TRANSIT := TRUE;
                _STATE := CRANE_STATES_T#CRANE_TURN_LEFT_NOT_METALLIC;
            END_IF;

        CRANE_STATES_T#CRANE_LIFT_MAGAZIN_METALLIC:
            _TRANSIT := FALSE;
            CRANELOWER := FALSE;
            IF CRANEUP THEN
                _TRANSIT := TRUE;
                _STATE := CRANE_STATES_T#CRANE_TURN_LEFT_METALLIC;
            END_IF;

        CRANE_STATES_T#CRANE_LIFT_NOT_METALLIC_BLACK:
            _TRANSIT := FALSE;
            CRANELOWER := FALSE;
            IF CRANEUP THEN
                _TRANSIT := TRUE;
                _STATE := CRANE_STATES_T#CRANE_TURN_LEFT_NOT_METALLIC_BLACK;
            END_IF;

        CRANE_STATES_T#CRANE_LOWER:
            _TRANSIT := FALSE;
            MAGAZINVACUUMON := TRUE;
            MAGAZINVACUUMOFF := FALSE;
            CRANELOWER := TRUE;
            IF CRANESUCKED THEN
                _TRANSIT := TRUE;
                _STATE := CRANE_STATES_T#STEP0;
            END_IF;

        CRANE_STATES_T#CRANE_ON_CONVEYOR:
            _TRANSIT := FALSE;
            CRANETURNCOUNTERCLOCKWISE := FALSE;
            CRANETURNCLOCKWISE := FALSE;
            CRANELOWER := TRUE;
            IF CRANEDOWN THEN
                _TRANSIT := TRUE;
                _STATE := CRANE_STATES_T#RELEASE;
            END_IF;

        CRANE_STATES_T#CRANE_ON_CONVEYOR_METALLIC:
            _TRANSIT := FALSE;
            CRANETURNCOUNTERCLOCKWISE := FALSE;
            CRANETURNCLOCKWISE := FALSE;
            CRANELOWER := TRUE;
            IF CRANEDOWN THEN
                _TRANSIT := TRUE;
                _STATE := CRANE_STATES_T#RELEASE;
            END_IF;

        CRANE_STATES_T#CRANE_ON_CONVEYOR_NOT_METALLICA_BLACK:
            _TRANSIT := FALSE;
            CRANETURNCOUNTERCLOCKWISE := FALSE;
            CRANETURNCLOCKWISE := FALSE;
            CRANELOWER := TRUE;
            IF CRANEDOWN THEN
                _TRANSIT := TRUE;
                _STATE := CRANE_STATES_T#RELEASE_BLACK;
            END_IF;

        CRANE_STATES_T#CRANE_ON_STAMP_METALLIC:
            _TRANSIT := FALSE;
            CRANETURNCOUNTERCLOCKWISE := FALSE;
            CRANETURNCLOCKWISE := FALSE;
            CRANELOWER := TRUE;
            IF CRANEDOWN THEN
                _TRANSIT := TRUE;
                _STATE := CRANE_STATES_T#RELEASE_WORKPIECE;
            END_IF;

        CRANE_STATES_T#CRANE_ON_STAMP_STOP_BLACK:
            _TRANSIT := FALSE;
            CRANETURNCLOCKWISE := FALSE;
            CRANETURNCOUNTERCLOCKWISE := FALSE;
            IF TRUE THEN
                _TRANSIT := TRUE;
                _STATE := CRANE_STATES_T#RESET_INTERCONNECT;
            END_IF;

        CRANE_STATES_T#CRANE_TURN_LEFT_BACK_TO_STAMP:
            _TRANSIT := FALSE;
            CRANETURNCOUNTERCLOCKWISE := TRUE;
            CRANETURNCLOCKWISE := FALSE;
            IF CRANEPOSITIONSTAMP THEN
                _TRANSIT := TRUE;
                _STATE := CRANE_STATES_T#CRANE_ON_STAMP_STOP_BLACK;
            END_IF;

        CRANE_STATES_T#CRANE_TURN_LEFT_FROM_STAMP:
            _TRANSIT := FALSE;
            CRANETURNCLOCKWISE := TRUE;
            CRANETURNCOUNTERCLOCKWISE := FALSE;
            IF CRANEONCONVEYOR THEN
                _TRANSIT := TRUE;
                _STATE := CRANE_STATES_T#CRANE_ON_CONVEYOR_METALLIC;
            END_IF;

        CRANE_STATES_T#CRANE_TURN_LEFT_METALLIC:
            _TRANSIT := FALSE;
            CRANETURNCOUNTERCLOCKWISE := TRUE;
            CRANETURNCLOCKWISE := FALSE;
            IF CRANEPOSITIONSTAMP THEN
                _TRANSIT := TRUE;
                _STATE := CRANE_STATES_T#CRANE_ON_STAMP_METALLIC;
            END_IF;

        CRANE_STATES_T#CRANE_TURN_LEFT_NOT_METALLIC:
            _TRANSIT := FALSE;
            CRANETURNCOUNTERCLOCKWISE := TRUE;
            CRANETURNCLOCKWISE := FALSE;
            IF CRANEONCONVEYOR THEN
                _TRANSIT := TRUE;
                _STATE := CRANE_STATES_T#CRANE_ON_CONVEYOR;
            END_IF;

        CRANE_STATES_T#CRANE_TURN_LEFT_NOT_METALLIC_BLACK:
            _TRANSIT := FALSE;
            CRANETURNCOUNTERCLOCKWISE := TRUE;
            CRANETURNCLOCKWISE := FALSE;
            IF CRANEONCONVEYOR THEN
                _TRANSIT := TRUE;
                _STATE := CRANE_STATES_T#CRANE_ON_CONVEYOR_NOT_METALLICA_BLACK;
            END_IF;

        CRANE_STATES_T#INIT:
            _TRANSIT := FALSE;
            IF TRUE THEN
                _TRANSIT := TRUE;
                _STATE := CRANE_STATES_T#START_CRANE;
            END_IF;

        CRANE_STATES_T#INTERSTEP:
            _TRANSIT := FALSE;
            STARTCOMMANDCRANE := TRUE;
            IF STARTVAR THEN
                _TRANSIT := TRUE;
                _STATE := CRANE_STATES_T#INTERSTEP_2;
            END_IF;

        CRANE_STATES_T#INTERSTEP_2:
            _TRANSIT := FALSE;
            IF SLIDERMOVEDOUT THEN
                _TRANSIT := TRUE;
                _STATE := CRANE_STATES_T#TIMEDELAY;
            END_IF;

        CRANE_STATES_T#LAST_WORKPIECE_AT_STAMP:
            _TRANSIT := FALSE;
            IF TRUE THEN
                _TRANSIT := TRUE;
                _STATE := CRANE_STATES_T#PAUSE;
            END_IF;

        CRANE_STATES_T#LOWER_CRANE:
            _TRANSIT := FALSE;
            CRANELOWER := TRUE;
            IF CRANEDOWN THEN
                _TRANSIT := TRUE;
                _STATE := CRANE_STATES_T#SUCK_AT_STAMP;
            END_IF;

        CRANE_STATES_T#MAGAZIN_STOP:
            _TRANSIT := FALSE;
            CRANETURNCLOCKWISE := FALSE;
            CRANETURNCOUNTERCLOCKWISE := FALSE;
            IF (NOT WORKPIECEREADY AND NOT STAMPSLIDERFILLED) THEN
                _TRANSIT := TRUE;
                _STATE := CRANE_STATES_T#NO_WORKPIECE_READY;
            ELSIF WORKPIECEREADY THEN
                _TRANSIT := TRUE;
                _STATE := CRANE_STATES_T#CRANE_LOWER;
            ELSIF (NOT WORKPIECEREADY AND STAMPSLIDERFILLED) THEN
                _TRANSIT := TRUE;
                _STATE := CRANE_STATES_T#LAST_WORKPIECE_AT_STAMP;
            END_IF;

        CRANE_STATES_T#MAGAZIN_STOP_BLACK:
            _TRANSIT := FALSE;
            CRANETURNCLOCKWISE := FALSE;
            CRANETURNCOUNTERCLOCKWISE := FALSE;
            MAGAZINVACUUMON := TRUE;
            MAGAZINVACUUMOFF := FALSE;
            CRANELOWER := TRUE;
            IF CRANESUCKED THEN
                _TRANSIT := TRUE;
                _STATE := CRANE_STATES_T#CRANE_LIFT_NOT_METALLIC_BLACK;
            END_IF;

        CRANE_STATES_T#NO_WORKPIECE_READY:
            _TRANSIT := FALSE;
            IF TRUE THEN
                _TRANSIT := TRUE;
                _STATE := CRANE_STATES_T#START_CRANE;
            END_IF;

        CRANE_STATES_T#RESET_INTERCONNECT:
            _TRANSIT := FALSE;
            INTERCONNECT := FALSE;
            TIMER1(IN := FALSE, PT := TIME#1MS);
            IF SLIDERMOVEDOUT THEN
                _TRANSIT := TRUE;
                _STATE := CRANE_STATES_T#LOWER_CRANE;
            END_IF;

        CRANE_STATES_T#START_CRANE:
            _TRANSIT := FALSE;
            CRANELOWER := FALSE;
            MAGAZINVACUUMOFF := TRUE;
            MAGAZINVACUUMON := FALSE;
            CRANETURNCOUNTERCLOCKWISE := FALSE;
            CRANETURNCLOCKWISE := FALSE;
            STARTVAR := FALSE;
            STARTCOMMANDCRANE := FALSE;
            IF (STARTBUTTONMAGAZIN = TRUE) THEN
                INTERCONNECTCRANESTARTCOMMAND := TRUE;
            END_IF;
            IF INTERCONNECTCRANESTARTCOMMAND THEN
                _TRANSIT := TRUE;
                _STATE := CRANE_STATES_T#CRANE_INIT;
            END_IF;

        CRANE_STATES_T#STEP0:
            _TRANSIT := FALSE;
            IF NOT MAGAZINCAPACITIVESENSOR THEN
                _TRANSIT := TRUE;
                _STATE := CRANE_STATES_T#CRANE_LIFT_MAGAZIN;
            ELSIF MAGAZINCAPACITIVESENSOR THEN
                _TRANSIT := TRUE;
                _STATE := CRANE_STATES_T#CRANE_LIFT_MAGAZIN_METALLIC;
            END_IF;

        CRANE_STATES_T#SUCK_AT_STAMP:
            _TRANSIT := FALSE;
            MAGAZINVACUUMON := TRUE;
            MAGAZINVACUUMOFF := FALSE;
            IF CRANESUCKED THEN
                _TRANSIT := TRUE;
                _STATE := CRANE_STATES_T#CRANE_LIFT_AT_STAMP;
            END_IF;

        CRANE_STATES_T#TIMEDELAY:
            _TRANSIT := FALSE;
            TIMEDELAY_TIMER(IN := TRUE, PT := TIMEDELAY_TIMER_DURATION);
            TIMEDELAY_TIMER_INTERCONNECT := TIMEDELAY_TIMER.Q;
            IF TIMEDELAY_TIMER_INTERCONNECT THEN
                _TRANSIT := TRUE;
                _STATE := CRANE_STATES_T#TURN_RIGHT;
            END_IF;

        CRANE_STATES_T#TURN_RIGHT:
            _TRANSIT := FALSE;
            CRANETURNCLOCKWISE := TRUE;
            CRANETURNCOUNTERCLOCKWISE := FALSE;
            IF CRANEONMAGAZIN THEN
                _TRANSIT := TRUE;
                _STATE := CRANE_STATES_T#MAGAZIN_STOP;
            END_IF;

        CRANE_STATES_T#TURN_RIGHT_BLACK:
            _TRANSIT := FALSE;
            CRANETURNCLOCKWISE := TRUE;
            CRANETURNCOUNTERCLOCKWISE := FALSE;
            IF CRANEONMAGAZIN THEN
                _TRANSIT := TRUE;
                _STATE := CRANE_STATES_T#MAGAZIN_STOP_BLACK;
            END_IF;

        CRANE_STATES_T#PAUSE:
            _TRANSIT := FALSE;
            TIMER1(IN := CRANEUP, PT := DURATION1);
            INTERCONNECT := TIMER1.Q;
            IF INTERCONNECT THEN
                _TRANSIT := TRUE;
                _STATE := CRANE_STATES_T#RESET_INTERCONNECT;
            END_IF;

        CRANE_STATES_T#RELEASE:
            _TRANSIT := FALSE;
            MAGAZINVACUUMOFF := TRUE;
            MAGAZINVACUUMON := FALSE;
            IF TRUE THEN
                _TRANSIT := TRUE;
                _STATE := CRANE_STATES_T#CRANE_LIFT_CONVEYOR;
            END_IF;

        CRANE_STATES_T#RELEASE_BLACK:
            _TRANSIT := FALSE;
            MAGAZINVACUUMON := FALSE;
            MAGAZINVACUUMOFF := TRUE;
            IF TRUE THEN
                _TRANSIT := TRUE;
                _STATE := CRANE_STATES_T#CRANE_LIFT_CONVEYOR_BLACK;
            END_IF;

        CRANE_STATES_T#RELEASE_WORKPIECE:
            _TRANSIT := FALSE;
            MAGAZINVACUUMOFF := TRUE;
            MAGAZINVACUUMON := FALSE;
            IF TRUE THEN
                _TRANSIT := TRUE;
                _STATE := CRANE_STATES_T#CRANE_GO_UP;
            END_IF;

            END_CASE;
END_PROGRAM

CONFIGURATION Config0
  RESOURCE Res0 ON PLC
    TASK TASK0(INTERVAL := T#50MS, PRIORITY := 0);
    PROGRAM INSTANCE0 WITH TASK0 : CRANE;
  END_RESOURCE
END_CONFIGURATION

(* ---- cycles.st ---- *)
PROGRAM CYCLES
    VAR_INPUT
    I : BOOL;
    END_VAR

    VAR
        MACRO : INT := 1;
        MICRO : INT := 1;
    END_VAR

    VAR_OUTPUT
        O : INT;
    END_VAR

    O := MACRO;
    MICRO := MICRO - 1;

    IF MICRO = 0 THEN
        MACRO := MACRO + 1;
        MICRO := MACRO;
    END_IF;
END_PROGRAM

CONFIGURATION Config0
  RESOURCE Res0 ON PLC
    TASK TASK0(INTERVAL := T#50MS, PRIORITY := 0);
    PROGRAM INSTANCE0 WITH TASK0 : CYCLES;
  END_RESOURCE
END_CONFIGURATION

(* ---- detwait.st ---- *)
PROGRAM DW
VAR_INPUT  I:INT; END_VAR
VAR_OUTPUT O:INT; END_VAR
VAR S : INT; END_VAR

S := S + 1;

IF I = 1 THEN
    O := 1;
ELSE
    O := S;
END_IF;

END_PROGRAM

CONFIGURATION Config0
  RESOURCE Res0 ON PLC
    TASK TASK0(INTERVAL := T#50MS, PRIORITY := 0);
    PROGRAM INSTANCE0 WITH TASK0 : DW;
  END_RESOURCE
END_CONFIGURATION

(* ---- detwait_long.st ---- *)
PROGRAM DW
VAR_INPUT  I:INT; END_VAR
VAR_OUTPUT O:INT; END_VAR
VAR S : INT; END_VAR

IF I = 0 THEN
    S := 0;
ELSIF I > 0 THEN
    S := S + 1;
END_IF;
O := S;
END_PROGRAM

CONFIGURATION Config0
  RESOURCE Res0 ON PLC
    TASK TASK0(INTERVAL := T#50MS, PRIORITY := 0);
    PROGRAM INSTANCE0 WITH TASK0 : DW;
  END_RESOURCE
END_CONFIGURATION

(* ---- detwait_wrong.st ---- *)
PROGRAM DW
VAR_INPUT  I:INT; END_VAR
VAR_OUTPUT O:INT; END_VAR
VAR S : INT; END_VAR

S := S + 1;
O := S;

END_PROGRAM

CONFIGURATION Config0
  RESOURCE Res0 ON PLC
    TASK TASK0(INTERVAL := T#50MS, PRIORITY := 0);
    PROGRAM INSTANCE0 WITH TASK0 : DW;
  END_RESOURCE
END_CONFIGURATION

(* ---- enum.st ---- *)
TYPE
    abc : (a, b, c);
END_TYPE

FUNCTION SEL_FB : abc
    VAR_INPUT
        a : BOOL;
        b,c : abc;
    END_VAR

    IF a THEN
        SEL_FB := b;
    ELSE
        SEL_FB := c;
    END_IF;
END_FUNCTION

PROGRAM ppp
    VAR i : INT; END_VAR
    VAR_OUTPUT o : abc; END_VAR

    o := SEL_FB(i = 0, abc#a, SEL_FB(i = 1, abc#b, abc#c));
    i := i + 1;
    i := SEL(i>2, 0, i);
END_PROGRAM

CONFIGURATION Config0
  RESOURCE Res0 ON PLC
    TASK task0(INTERVAL := T#50ms, PRIORITY := 0);
    PROGRAM instance0 WITH task0 : ppp;
  END_RESOURCE
END_CONFIGURATION

(* ---- expressionVisitorTest.basicTest.st ---- *)
TYPE
    MY_ENUM : (POSSIBLE, VALUES, ENUM);
END_TYPE

PROGRAM MY_STH
    VAR_INPUT
        ACTIVE : BOOL := TRUE;
        NUMBER : INT := 1;
        MY_ENUM_1 : MY_ENUM;
    END_VAR

    VAR_OUTPUT
        MY_OUTPUT : MY_ENUM;
        SERIOUSLY : BOOL;
    END_VAR

    VAR
        MY_ENUM_LOCAL : MY_ENUM;
    END_VAR

    VAR_IN_OUT
        ACTIVE_INOUT : BOOL;
    END_VAR

   SERIOUSLY := NOT FALSE;
   NUMBER := (- 19);
   NUMBER := 1 + 2;

END_PROGRAM

CONFIGURATION Config0
  RESOURCE Res0 ON PLC
    TASK TASK0(INTERVAL := T#50MS, PRIORITY := 0);
    PROGRAM INSTANCE0 WITH TASK0 : MY_STH;
  END_RESOURCE
END_CONFIGURATION

(* ---- history.st ---- *)
PROGRAM constantprogram
    VAR_INPUT
        i : INT;
    END_VAR

    VAR
        a,b,c,d : INT;
    END_VAR

    VAR_OUTPUT
        o : INT;
    END_VAR

    o := d;
    d := c;
    c := b;
    b := a;
    a := i;

END_PROGRAM

CONFIGURATION Config0
  RESOURCE Res0 ON PLC
    TASK task0(INTERVAL := T#50ms, PRIORITY := 0);
    PROGRAM instance0 WITH task0 : constantprogram;
  END_RESOURCE
END_CONFIGURATION

(* ---- ifac1.st ---- *)
TYPE
  OPMODE : (OP , TEACH);
  TEACHSTATUS :  (OK, NOTEACHPOINTS, TEACHING, INVALIDTEACHPOINTS, INVALIDINPUTVALUE);
END_TYPE

PROGRAM ANALOGSENSOR

VAR CONSTANT
  SENSORINPUT_MIN : INT := 0;
  SENSORINPUT_MAX : INT := 4095;
  TEACHTIMEOUT : TIME := TIME#20S0MS;
  ICONST : INT := 1000;
END_VAR

VAR_INPUT
  TPSET, SENSORINPUT, TPY  : INT;
  OPERATIONMODE : OPMODE;
END_VAR

VAR_OUTPUT
  SENSOROUTPUT : INT;
END_VAR

VAR
  INITIAL          : BOOL;
  LASTMODE : OPMODE;
  STATUS        : TEACHSTATUS;
  TEACHSTEP : SINT;
  X_TEMP, Y_TEMP, T, M, X1, Y1, X2, Y2 : INT;

  TIMEOUT : TON;
END_VAR

IF NOT INITIAL THEN
  X1 := 0;
  Y1 := 0;
  X2 := 0;
  Y2 := 0;
  STATUS := TEACHSTATUS#NOTEACHPOINTS;
  INITIAL := TRUE;
ELSE
  IF OPERATIONMODE = OPMODE#OP THEN
    IF STATUS = TEACHSTATUS#OK AND SENSORINPUT >= SENSORINPUT_MIN AND SENSORINPUT <= SENSORINPUT_MAX THEN
      SENSOROUTPUT := M * SENSORINPUT / ICONST + T;
    ELSE
      SENSOROUTPUT := 0;
    END_IF;
  ELSIF OPERATIONMODE = OPMODE#TEACH THEN
    IF LASTMODE <> OPERATIONMODE THEN
      TEACHSTEP := 0;
      TIMEOUT(IN := FALSE);
    END_IF;

    CASE TEACHSTEP OF
      0:
         STATUS := TEACHSTATUS#TEACHING;
         TIMEOUT(IN := TRUE, PT:=TEACHTIMEOUT);
         IF TIMEOUT.Q THEN
           OPERATIONMODE := OPMODE#OP;
         END_IF;

         IF INT_TO_BOOL(TPSET) AND SENSORINPUT >= SENSORINPUT_MIN AND SENSORINPUT <= SENSORINPUT_MAX THEN
           Y1 := TPY;
           X1 := SENSORINPUT;
           TEACHSTEP := 1;
           TIMEOUT(IN := FALSE);
         END_IF;
      1:
         IF INT_TO_BOOL(TPSET) = FALSE THEN
           TEACHSTEP := 2;
         END_IF;
      2:
         TIMEOUT(IN := TRUE, PT:=TEACHTIMEOUT);

         IF TIMEOUT.Q THEN
           OPERATIONMODE := OPMODE#OP;
         END_IF;

         IF INT_TO_BOOL(TPSET) AND SENSORINPUT >= SENSORINPUT_MIN AND SENSORINPUT <= SENSORINPUT_MAX THEN
           Y2 := TPY;
           X2 := SENSORINPUT;
           TEACHSTEP := 3;
           TIMEOUT(IN := FALSE);
         END_IF;
       3:
        IF X1 > X2 THEN
           X_TEMP := X1;
	   Y_TEMP := Y1;
	   X1 := X2;
	   Y1 := Y2;
	   X2 := X_TEMP;
	   Y2 := Y_TEMP;
         END_IF;

         IF X2 - X1 <> 0 THEN
           M   := (Y2 - Y1) * ICONST / (X2 - X1);
           T   := Y1 - M * X1 / ICONST;
           STATUS := TEACHSTATUS#OK;
	 ELSE
           STATUS := TEACHSTATUS#INVALIDTEACHPOINTS;
	   OPERATIONMODE := OPMODE#OP;
         END_IF;
       END_CASE;
  END_IF;
END_IF;
LASTMODE := OPERATIONMODE;
END_PROGRAM

CONFIGURATION Config0
  RESOURCE Res0 ON PLC
    TASK TASK0(INTERVAL := T#50MS, PRIORITY := 0);
    PROGRAM INSTANCE0 WITH TASK0 : ANALOGSENSOR;
  END_RESOURCE
END_CONFIGURATION

(* ---- lr.new.overflow.st ---- *)
TYPE
  OPMODE : (OP , TEACH);
  TEACHSTATUS :  (OK, NOTEACHPOINTS, TEACHING, INVALIDTEACHPOINTS, INVALIDINPUTVALUE);
END_TYPE

PROGRAM  ANALOGSENSOR

VAR CONSTANT
  SENSORINPUT_MIN : INT := 0;
  SENSORINPUT_MAX : INT := 4095;
  TEACHTIMEOUT : TIME := TIME#20S0MS;
  ICONST : INT := 1000;
END_VAR

VAR_INPUT
  TPSET : BOOL;
  SENSORINPUT, TPY  : INT;
  OPERATIONMODE : OPMODE;
END_VAR

VAR_OUTPUT
  SENSOROUTPUT : INT;
END_VAR

VAR
  INITIAL          : BOOL;
  LASTMODE         : OPMODE;
  STATUS           : TEACHSTATUS;
  TEACHSTEP        : INT;
  X_TEMP, Y_TEMP, T, M, X1, Y1, X2, Y2 : INT;
  TIMEOUT          : TON;
END_VAR

IF NOT INITIAL THEN
  X1 := 0;
  Y1 := 0;
  X2 := 0;
  Y2 := 0;
  STATUS := TEACHSTATUS#NOTEACHPOINTS;
  INITIAL := TRUE;
ELSE
  IF OPERATIONMODE = OPMODE#OP THEN
    IF STATUS = TEACHSTATUS#OK AND SENSORINPUT >= SENSORINPUT_MIN AND SENSORINPUT <= SENSORINPUT_MAX THEN
      SENSOROUTPUT := M * SENSORINPUT / ICONST + T;
    ELSE
      SENSOROUTPUT := 0;
    END_IF;
  ELSIF OPERATIONMODE = OPMODE#TEACH THEN
    IF LASTMODE <> OPERATIONMODE THEN
      TEACHSTEP := 0;
      TIMEOUT(IN := FALSE);
    END_IF;

    CASE TEACHSTEP OF
      0:
         STATUS := TEACHSTATUS#TEACHING;
         TIMEOUT(IN := TRUE, PT:=TEACHTIMEOUT);
         IF TIMEOUT.Q THEN
           OPERATIONMODE := OPMODE#OP;
         END_IF;

         IF TPSET AND SENSORINPUT >= SENSORINPUT_MIN AND SENSORINPUT <= SENSORINPUT_MAX THEN
           Y1 := TPY;
           X1 := SENSORINPUT;
           TEACHSTEP := 1;
           TIMEOUT(IN := FALSE);
         END_IF;
      1:
         IF TPSET = FALSE THEN
           TEACHSTEP := 2;
         END_IF;
      2:
         TIMEOUT(IN := TRUE, PT:=TEACHTIMEOUT);

         IF TIMEOUT.Q THEN
           OPERATIONMODE := OPMODE#OP;
         END_IF;

         IF TPSET AND SENSORINPUT >= SENSORINPUT_MIN
             AND SENSORINPUT <= SENSORINPUT_MAX THEN
           Y2 := TPY;
           X2 := SENSORINPUT;
           TEACHSTEP := 3;
           TIMEOUT(IN := FALSE);
         END_IF;
       3:
        IF X1 > X2 THEN
           X_TEMP := X1;
	   Y_TEMP := Y1;
	   X1 := X2;
	   Y1 := Y2;
	   X2 := X_TEMP;
	   Y2 := Y_TEMP;
         END_IF;

         IF X2 - X1 <> 0 THEN
           M   := (Y2 - Y1) * ICONST / (X1 - X2);
           T   := (M * X1 / ICONST) - Y1;
           STATUS := TEACHSTATUS#OK;
	 ELSE
           STATUS := TEACHSTATUS#INVALIDTEACHPOINTS;
	   OPERATIONMODE := OPMODE#OP;
         END_IF;
       END_CASE;
  END_IF;
END_IF;
LASTMODE := OPERATIONMODE;
END_PROGRAM

CONFIGURATION Config0
  RESOURCE Res0 ON PLC
    TASK TASK0(INTERVAL := T#50MS, PRIORITY := 0);
    PROGRAM INSTANCE0 WITH TASK0 : ANALOGSENSOR;
  END_RESOURCE
END_CONFIGURATION

(* ---- lr.new.st ---- *)
TYPE
  OPMODE : (OP , TEACH);
  TEACHSTATUS :  (OK, NOTEACHPOINTS, TEACHING, INVALIDTEACHPOINTS, INVALIDINPUTVALUE);
END_TYPE

PROGRAM  ANALOGSENSOR

VAR CONSTANT
  SENSORINPUT_MIN : INT := 0;
  SENSORINPUT_MAX : INT := 4095;
  TEACHTIMEOUT : TIME := TIME#20S0MS;
  ICONST : INT := 1000;
END_VAR

VAR_INPUT
  TPSET : BOOL;
  SENSORINPUT, TPY  : INT;
  OPERATIONMODE : OPMODE;
END_VAR

VAR_OUTPUT
  SENSOROUTPUT : INT;
END_VAR

VAR
  INITIAL          : BOOL;
  LASTMODE         : OPMODE;
  STATUS           : TEACHSTATUS;
  TEACHSTEP        : INT;
  X_TEMP, Y_TEMP, T, M, X1, Y1, X2, Y2 : INT;
  TIMEOUT          : TON;
END_VAR

IF NOT INITIAL THEN
  X1 := 0;
  Y1 := 0;
  X2 := 0;
  Y2 := 0;
  STATUS := TEACHSTATUS#NOTEACHPOINTS;
  INITIAL := TRUE;
ELSE
  IF OPERATIONMODE = OPMODE#OP THEN
    IF STATUS = TEACHSTATUS#OK AND SENSORINPUT >= SENSORINPUT_MIN AND SENSORINPUT <= SENSORINPUT_MAX THEN
      SENSOROUTPUT := M * SENSORINPUT / ICONST + T;
    ELSE
      SENSOROUTPUT := 0;
    END_IF;
  ELSIF OPERATIONMODE = OPMODE#TEACH THEN
    IF LASTMODE <> OPERATIONMODE THEN
      TEACHSTEP := 0;
      TIMEOUT(IN := FALSE);
    END_IF;

    CASE TEACHSTEP OF
      0:
         STATUS := TEACHSTATUS#TEACHING;
         TIMEOUT(IN := TRUE, PT:=TEACHTIMEOUT);
         IF TIMEOUT.Q THEN
           OPERATIONMODE := OPMODE#OP;
         END_IF;

         IF TPSET AND SENSORINPUT >= SENSORINPUT_MIN AND SENSORINPUT <= SENSORINPUT_MAX THEN
           Y1 := TPY;
           X1 := SENSORINPUT;
           TEACHSTEP := 1;
           TIMEOUT(IN := FALSE);
         END_IF;
      1:
         IF TPSET = FALSE THEN
           TEACHSTEP := 2;
         END_IF;
      2:
         TIMEOUT(IN := TRUE, PT:=TEACHTIMEOUT);

         IF TIMEOUT.Q THEN
           OPERATIONMODE := OPMODE#OP;
         END_IF;

         IF TPSET AND SENSORINPUT >= SENSORINPUT_MIN
             AND SENSORINPUT <= SENSORINPUT_MAX THEN
           Y2 := TPY;
           X2 := SENSORINPUT;
           TEACHSTEP := 3;
           TIMEOUT(IN := FALSE);
         END_IF;
       3:
        IF X1 > X2 THEN
           X_TEMP := X1;
	   Y_TEMP := Y1;
	   X1 := X2;
	   Y1 := Y2;
	   X2 := X_TEMP;
	   Y2 := Y_TEMP;
         END_IF;

         IF X2 - X1 <> 0 THEN
           M   := (Y2 - Y1) * ICONST / (X2 - X1);
           T   := Y1 - M * X1 / ICONST;
           STATUS := TEACHSTATUS#OK;
	 ELSE
           STATUS := TEACHSTATUS#INVALIDTEACHPOINTS;
	   OPERATIONMODE := OPMODE#OP;
         END_IF;
       END_CASE;
  END_IF;
END_IF;
LASTMODE := OPERATIONMODE;
END_PROGRAM

CONFIGURATION Config0
  RESOURCE Res0 ON PLC
    TASK TASK0(INTERVAL := T#50MS, PRIORITY := 0);
    PROGRAM INSTANCE0 WITH TASK0 : ANALOGSENSOR;
  END_RESOURCE
END_CONFIGURATION

(* ---- lr.new2.st ---- *)
TYPE
  OPMODE : (OP , TEACH);
  TEACHSTATUS :  (OK, NOTEACHPOINTS, TEACHING, INVALIDTEACHPOINTS, INVALIDINPUTVALUE);
END_TYPE

PROGRAM ANALOGSENSOR

VAR
  SENSORINPUT_MIN : INT := 0;
  SENSORINPUT_MAX : INT := 4095;
  TEACHTIMEOUT : TIME := TIME#20S0MS;
  ICONST : INT := 1000;
END_VAR

VAR_INPUT
  TPSET : BOOL;
  SENSORINPUT, TPY  : INT;
  OPERATIONMODE : OPMODE;
END_VAR

VAR_OUTPUT
  SENSOROUTPUT : INT;
END_VAR

VAR
  INITIAL          : BOOL;
  LASTMODE         : OPMODE;
  STATUS           : TEACHSTATUS;
  TEACHSTEP        : INT;
  X_TEMP, Y_TEMP, T, M, X1, Y1, X2, Y2 : INT;
  TIMEOUT          : TON;
END_VAR

IF NOT INITIAL THEN
  X1 := 0;
  Y1 := 0;
  X2 := 0;
  Y2 := 0;
  STATUS := TEACHSTATUS#NOTEACHPOINTS;
  INITIAL := TRUE;
ELSE
  IF OPERATIONMODE = OPMODE#OP THEN
    IF STATUS = TEACHSTATUS#OK AND SENSORINPUT >= SENSORINPUT_MIN AND SENSORINPUT <= SENSORINPUT_MAX THEN
      SENSOROUTPUT := M * SENSORINPUT / ICONST + T;
    ELSE
      SENSOROUTPUT := 0;
    END_IF;
  ELSIF OPERATIONMODE = OPMODE#TEACH THEN
    IF LASTMODE <> OPERATIONMODE THEN
      TEACHSTEP := 0;
      TIMEOUT(IN := FALSE);
    END_IF;

    CASE TEACHSTEP OF
      0:
         STATUS := TEACHSTATUS#TEACHING;
         TIMEOUT(IN := TRUE, PT:=TEACHTIMEOUT);
         IF TIMEOUT.Q THEN
           OPERATIONMODE := OPMODE#OP;
         END_IF;

         IF TPSET AND SENSORINPUT >= SENSORINPUT_MIN AND SENSORINPUT <= SENSORINPUT_MAX THEN
           Y1 := TPY;
           X1 := SENSORINPUT;
           TEACHSTEP := 1;
           TIMEOUT(IN := FALSE);
         END_IF;
      1:
         IF TPSET = FALSE THEN
           TEACHSTEP := 2;
         END_IF;
      2:
         TIMEOUT(IN := TRUE, PT:=TEACHTIMEOUT);

         IF TIMEOUT.Q THEN
           OPERATIONMODE := OPMODE#OP;
         END_IF;

         IF TPSET AND SENSORINPUT >= SENSORINPUT_MIN
             AND SENSORINPUT <= SENSORINPUT_MAX THEN
           Y2 := TPY;
           X2 := SENSORINPUT;
           TEACHSTEP := 3;
           TIMEOUT(IN := FALSE);
         END_IF;
       3:
        IF X1 > X2 THEN
           X_TEMP := X1;
	   Y_TEMP := Y1;
	   X1 := X2;
	   Y1 := Y2;
	   X2 := X_TEMP;
	   Y2 := Y_TEMP;
         END_IF;

         IF X2 - X1 <> 0 THEN
           M   := (Y1 - Y2) * ICONST / (X2 - X1);
           T   := M * X1 / ICONST - Y1;
           STATUS := TEACHSTATUS#OK;
	 ELSE
           STATUS := TEACHSTATUS#INVALIDTEACHPOINTS;
	   OPERATIONMODE := OPMODE#OP;
         END_IF;
       END_CASE;
  END_IF;
END_IF;
LASTMODE := OPERATIONMODE;
END_PROGRAM

CONFIGURATION Config0
  RESOURCE Res0 ON PLC
    TASK TASK0(INTERVAL := T#50MS, PRIORITY := 0);
    PROGRAM INSTANCE0 WITH TASK0 : ANALOGSENSOR;
  END_RESOURCE
END_CONFIGURATION

(* ---- lr.st ---- *)
TYPE
  OPMODE : (OP , TEACH);
  TEACHSTATUS :  (OK, NOTEACHPOINTS, TEACHING, INVALIDTEACHPOINTS, INVALIDINPUTVALUE);
END_TYPE

PROGRAM  ANALOGSENSOR

VAR CONSTANT
  SENSORINPUT_MIN : INT := 0;
  SENSORINPUT_MAX : INT := 4095;
  TEACHTIMEOUT : TIME := TIME#20S0MS;
  ICONST : INT := 1000;
END_VAR

VAR_INPUT
  TPSET : BOOL;
  SENSORINPUT, TPY  : INT;
  OPERATIONMODE : OPMODE;
END_VAR

VAR_OUTPUT
  SENSOROUTPUT : INT;
END_VAR

VAR
  INITIAL          : BOOL;
  LASTMODE         : OPMODE;
  STATUS           : TEACHSTATUS;
  TEACHSTEP        : INT;
  X_TEMP, Y_TEMP, T, M, X1, Y1, X2, Y2 : INT;
  TIMEOUT          	: TON;
END_VAR

IF NOT INITIAL THEN
  X1 := 0;
  Y1 := 0;
  X2 := 0;
  Y2 := 0;
  STATUS := TEACHSTATUS#NOTEACHPOINTS;
  INITIAL := TRUE;
ELSE
  IF OPERATIONMODE = OPMODE#OP THEN
    IF STATUS = TEACHSTATUS#OK AND SENSORINPUT >= SENSORINPUT_MIN AND SENSORINPUT <= SENSORINPUT_MAX THEN
      SENSOROUTPUT := M * SENSORINPUT / ICONST + T;
    ELSE
      SENSOROUTPUT := 0;
    END_IF;
  ELSIF OPERATIONMODE = OPMODE#TEACH THEN
    IF LASTMODE <> OPERATIONMODE THEN
      TEACHSTEP := 0;
      TIMEOUT(IN := FALSE);
    END_IF;

    CASE TEACHSTEP OF
      0:
         STATUS := TEACHSTATUS#TEACHING;
         TIMEOUT(IN := TRUE, PT:=TEACHTIMEOUT);
         IF TIMEOUT.Q THEN
           OPERATIONMODE := OPMODE#OP;
         END_IF;

         IF TPSET AND SENSORINPUT >= SENSORINPUT_MIN AND SENSORINPUT <= SENSORINPUT_MAX THEN
           Y1 := TPY;
           X1 := SENSORINPUT;
           TEACHSTEP := 1;
           TIMEOUT(IN := FALSE);
         END_IF;
      1:
         IF TPSET = FALSE THEN
           TEACHSTEP := 2;
         END_IF;
      2:
         TIMEOUT(IN := TRUE, PT:=TEACHTIMEOUT);

         IF TIMEOUT.Q THEN
           OPERATIONMODE := OPMODE#OP;
         END_IF;

         IF TPSET AND SENSORINPUT >= SENSORINPUT_MIN
             AND SENSORINPUT <= SENSORINPUT_MAX THEN
           Y2 := TPY;
           X2 := SENSORINPUT;
           TEACHSTEP := 3;
           TIMEOUT(IN := FALSE);
         END_IF;
       3:
        IF X1 > X2 THEN
           X_TEMP := X1;
	   Y_TEMP := Y1;
	   X1 := X2;
	   Y1 := Y2;
	   X2 := X_TEMP;
	   Y2 := Y_TEMP;
         END_IF;

         IF X2 - X1 <> 0 THEN
           M   := (Y2 - Y1) * ICONST / (X2 - X1);
           T   := Y1 - M * X1 / ICONST;
           STATUS := TEACHSTATUS#OK;
	 ELSE
           STATUS := TEACHSTATUS#INVALIDTEACHPOINTS;
	   OPERATIONMODE := OPMODE#OP;
         END_IF;
       END_CASE;
  END_IF;
END_IF;
  LASTMODE := OPERATIONMODE;
END_PROGRAM
CONFIGURATION Config0
  RESOURCE Res0 ON PLC
    TASK TASK0(INTERVAL := T#50MS, PRIORITY := 0);
    PROGRAM INSTANCE0 WITH TASK0 : ANALOGSENSOR;
  END_RESOURCE
END_CONFIGURATION

(* ---- MinMax.st ---- *)
TYPE
  OPERATIONMODE : (LEARN , ACTIVE);
END_TYPE

FUNCTION SEL : INT
VAR_INPUT
        G : BOOL;
        A,B : INT;
END_VAR

IF G THEN SEL := A;
     ELSE SEL := B; END_IF;

END_FUNCTION

FUNCTION MAX : INT
VAR_INPUT
        IN0 : INT;
        IN1 : INT;
END_VAR

MAX := SEL(IN0>=IN1, IN0, IN1);

END_FUNCTION

FUNCTION MIN : INT
VAR_INPUT
        IN0 : INT;
        IN1 : INT;
END_VAR

MIN := SEL(IN0<=IN1, IN0, IN1);

END_FUNCTION

PROGRAM MINMAX

VAR CONSTANT
    WAIT_BEFORE_WARNING : INT := 3; (*   AMOUNT OF CYCLES OUTSIDE  BEFORE GIVEN A WARNING.*)
    WAIT_AFTER_WARNING  : INT := 3; (*   AMOUNT OF CYCLES INSIDE, BEFORE WITHDRAW WARNING.*)
END_VAR

VAR_INPUT
  MODE     : OPERATIONMODE; (* LEARNING OR ACTIVE MODE *)
  LEARN    : BOOL;          (* TRUE IFF CURRENT SIGNAL SHOULD BE LEARNT *)
   I        : INT;           (* INPUT SIGNAL*)
 END_VAR

VAR_OUTPUT
        W       : BOOL;     (* WARNING FLAG, IFF _I \NOT\IN [LOWER,UPPER]_*)
        Q       : INT;      (* TRUNCATED INPUT SIGNAL*)
END_VAR

VAR
        LOWER : INT :=  32766;  (* MINIMAL TEACHED VALUE*)
        UPPER : INT := -32767;  (* MAXIMAL TEACH VALUE*)
        CNTQUENCH : INT := 3;   (* REMAINING CYCLES FOR WITHDRAW WARNING*)
        CNTHEAT   : INT := 3;   (* REMAINING CYCLES TO SIGNAL WARNING*)
 END_VAR

IF MODE = OPERATIONMODE#LEARN THEN (* GO INTO LEARNING*)
        IF LEARN THEN
                LOWER := MIN(LOWER, I);
                UPPER := MAX(UPPER, I);
        END_IF;
        Q := 0;
        W := FALSE;
ELSE
        IF UPPER < LOWER THEN
                Q := 0;
                W := TRUE;
        ELSE
                Q := MIN( UPPER, MAX( LOWER, I) );
                IF I <> Q THEN
                        CNTHEAT := CNTHEAT - 1;
                        CNTQUENCH := WAIT_AFTER_WARNING;
                        IF CNTHEAT = 0 THEN
                                W := TRUE;
                        END_IF;
                ELSE
                        CNTQUENCH := CNTQUENCH - 1;
                        CNTHEAT := WAIT_BEFORE_WARNING;
                        IF CNTQUENCH = 0 THEN
                                W := FALSE;
                        END_IF;
                END_IF;
         END_IF;
END_IF;

END_PROGRAM

CONFIGURATION Config0
  RESOURCE Res0 ON PLC
    TASK TASK0(INTERVAL := T#50MS, PRIORITY := 0);
    PROGRAM INSTANCE0 WITH TASK0 : MINMAX;
  END_RESOURCE
END_CONFIGURATION

(* ---- OneCnt.st ---- *)
PROGRAM OneCnt
VAR s : INT; END_VAR

VAR_OUTPUT
    c : INT;
END_VAR

    s := s + 1;
    c :=  s;

END_PROGRAM

CONFIGURATION Config0
  RESOURCE Res0 ON PLC
    TASK task0(INTERVAL := T#50ms, PRIORITY := 0);
    PROGRAM instance0 WITH task0 : OneCnt;
  END_RESOURCE
END_CONFIGURATION

(* ---- OneIncrement.st ---- *)
PROGRAM STEPS

VAR_OUTPUT O : INT := 0; END_VAR

O := O + 1;

END_PROGRAM

CONFIGURATION Config0
  RESOURCE Res0 ON PLC
    TASK TASK0(INTERVAL := T#50MS, PRIORITY := 0);
    PROGRAM INSTANCE0 WITH TASK0 : STEPS;
  END_RESOURCE
END_CONFIGURATION

(* ---- runtimeTest.advancedTest_wMan.st ---- *)
TYPE
    TRAFFICLIGHT : (RED, GREEN);
END_TYPE

PROGRAM PEDESTRIANTRAFFICLIGHT

    VAR_INPUT
        PEDBTNPRESS : BOOL := TRUE;
    END_VAR

    VAR_OUTPUT
        CARLIGHT : TRAFFICLIGHT;
        PEDLIGHT : TRAFFICLIGHT;
        COUNTER : INT := 50;
    END_VAR

    VAR
        BUTTONPRESSEDBEFORE : BOOL := FALSE;
    END_VAR

    IF (NOT BUTTONPRESSEDBEFORE) AND PEDBTNPRESS THEN
        CARLIGHT := TRAFFICLIGHT#RED;
    END_IF;

    IF COUNTER = 10 THEN
        PEDLIGHT := TRAFFICLIGHT#GREEN;
    ELSIF COUNTER = 40 THEN
     PEDLIGHT := TRAFFICLIGHT#RED;
    ELSIF COUNTER = 50 THEN
        CARLIGHT := TRAFFICLIGHT#GREEN;
    END_IF;

    IF CARLIGHT = TRAFFICLIGHT#RED THEN
        COUNTER := COUNTER + 1;
    ELSE
        COUNTER := 0;
    END_IF;

    BUTTONPRESSEDBEFORE := PEDBTNPRESS;

END_PROGRAM

CONFIGURATION Config0
  RESOURCE Res0 ON PLC
    TASK TASK0(INTERVAL := T#50MS, PRIORITY := 0);
    PROGRAM INSTANCE0 WITH TASK0 : PEDESTRIANTRAFFICLIGHT;
  END_RESOURCE
END_CONFIGURATION

(* ---- runtimeTest.cycles.st ---- *)
PROGRAM MY_STH
    VAR_INPUT
        I : INT;
    END_VAR

    VAR
        COUNTER : INT := 0;
    END_VAR

   COUNTER := COUNTER + I;

   IF COUNTER > 1000 THEN
        COUNTER := 0;
   END_IF;

END_PROGRAM

CONFIGURATION Config0
  RESOURCE Res0 ON PLC
    TASK TASK0(INTERVAL := T#50MS, PRIORITY := 0);
    PROGRAM INSTANCE0 WITH TASK0 : MY_STH;
  END_RESOURCE
END_CONFIGURATION

(* ---- runtimeTest.elevatorTest.st ---- *)
TYPE
  MOTOR_STATE : (GoDown, Stationary, GoUp);
  DOOR_STATE : (Open, Closed);
END_TYPE

PROGRAM Elevator

  VAR_INPUT
    CurrentPos : INT := 3;
    RequestedPos : INT := 5;
    ButtonPressed : BOOL;
  END_VAR

  VAR_OUTPUT
    Motor : MOTOR_STATE := MOTOR_STATE#Stationary;
    Door : DOOR_STATE := DOOR_STATE#Open;
  END_VAR

  IF ButtonPressed THEN

    Door := DOOR_STATE#Closed;

    IF RequestedPos > CurrentPos THEN
      Motor := MOTOR_STATE#GoUp;
    ELSIF RequestedPos < CurrentPos THEN
      Motor := MOTOR_STATE#GoDown;
    END_IF;

  END_IF;

  IF RequestedPos = CurrentPos THEN
    Motor := MOTOR_STATE#Stationary;
    Door := DOOR_STATE#Open;
  END_IF;

END_PROGRAM
CONFIGURATION Config0
  RESOURCE Res0 ON PLC
    TASK task0(INTERVAL := T#50ms, PRIORITY := 0);
    PROGRAM instance0 WITH task0 : Elevator;
  END_RESOURCE
END_CONFIGURATION

(* ---- runtimeTest.enumTest.st ---- *)
TYPE
    MY_ENUM : (POSSIBLE, VALUES, ENUM);
END_TYPE

PROGRAM MY_STH
    VAR_INPUT
        ACTIVE : BOOL := TRUE;
        NUMBER : INT := 1;
        MY_ENUM_1 : MY_ENUM;
    END_VAR

   ACTIVE := NOT FALSE;
   NUMBER := (- 19);
   NUMBER := NUMBER + 2;
   ACTIVE := NOT ACTIVE;
   NUMBER := 3;

   IF NUMBER = 3 THEN
    NUMBER :=300;
   END_IF;
END_PROGRAM

CONFIGURATION Config0
  RESOURCE Res0 ON PLC
    TASK TASK0(INTERVAL := T#50MS, PRIORITY := 0);
    PROGRAM INSTANCE0 WITH TASK0 : MY_STH;
  END_RESOURCE
END_CONFIGURATION

(* ---- runtimeTest.forLoopTest.st ---- *)
PROGRAM MY_STH
    VAR_INPUT
        VAR1 : INT := 2;
        VAR2 : INT := 0;
        COUNTER2 : INT := 0;
    END_VAR

   FOR COUNTER2:=1 TO 5 DO
       VAR1:=VAR1*2;
   END_FOR;

   FOR COUNTER2:=1 TO 5 DO
      VAR2:=VAR2+1;
   END_FOR;
END_PROGRAM

CONFIGURATION Config0
  RESOURCE Res0 ON PLC
    TASK TASK0(INTERVAL := T#50MS, PRIORITY := 0);
    PROGRAM INSTANCE0 WITH TASK0 : MY_STH;
  END_RESOURCE
END_CONFIGURATION

(* ---- runtimeTest.functionTest.st ---- *)
FUNCTION FuncAdd : REAL
VAR_INPUT
  a: REAL;
  b: REAL;
END_VAR

FuncAdd := INT_TO_REAL(2)*a - INT_TO_REAL(22)*b;
END_FUNCTION

PROGRAM my_sth
VAR_INPUT
  Var1 : REAL := REAL#2.0;
  x : REAL := REAL#7.0;
  y : REAL := REAL#8.0;
END_VAR

Var1 := FuncAdd(x, y);
END_PROGRAM

CONFIGURATION Config0
  RESOURCE Res0 ON PLC
    TASK task0(INTERVAL := T#50ms, PRIORITY := 0);
    PROGRAM instance0 WITH task0 : my_sth;
  END_RESOURCE
END_CONFIGURATION

(* ---- runtimeTest.repeatLoopTest.st ---- *)
PROGRAM MY_STH
    VAR_INPUT
        VAR1 : INT := 2;
        COUNTER : INT := 4;
    END_VAR

   REPEAT
       VAR1 := VAR1*2;
       COUNTER := COUNTER-1;
   UNTIL
       COUNTER=0
   END_REPEAT;
END_PROGRAM

CONFIGURATION Config0
  RESOURCE Res0 ON PLC
    TASK TASK0(INTERVAL := T#50MS, PRIORITY := 0);
    PROGRAM INSTANCE0 WITH TASK0 : MY_STH;
  END_RESOURCE
END_CONFIGURATION

(* ---- runtimeTest.structTest_wMan.st ---- *)
TYPE
    POINT: STRUCT
        X: INT;
        Y: INT;
    END_STRUCT;
END_TYPE

PROGRAM MY_STH
    VAR
        VAR1 : POINT;
        VAR2 : INT;
        VAR3 : POINT := (X:= 1, Y:=2);
    END_VAR

    VAR2 := 7;
    VAR1.X := 1;
    VAR1.Y := 2;
    VAR3.Y := 100;
    VAR3.Y := -7000; (* ORIGINAL NUMBER IS -70000, CAN'T COMPILE FROM OPENPLC*)

END_PROGRAM

CONFIGURATION Config0
  RESOURCE Res0 ON PLC
    TASK TASK0(INTERVAL := T#50MS, PRIORITY := 0);
    PROGRAM INSTANCE0 WITH TASK0 : MY_STH;
  END_RESOURCE
END_CONFIGURATION

(* ---- runtimeTest.testIfStatement.st ---- *)
PROGRAM my_sth
    VAR_INPUT
        number : INT := 1;
        n2 : INT;
        active : BOOL := True;
    END_VAR

   number := 3;

   if number = 3 THEN
    number :=300;
   END_IF;

   if active THEN
    n2 := 4;
    END_IF;
END_PROGRAM

CONFIGURATION Config0
  RESOURCE Res0 ON PLC
    TASK task0(INTERVAL := T#50ms, PRIORITY := 0);
    PROGRAM instance0 WITH task0 : my_sth;
  END_RESOURCE
END_CONFIGURATION

(* ---- runtimeTest.testVariableReference.st ---- *)
PROGRAM my_sth
    VAR_INPUT
        b : BOOL := True;
        b2 : BOOL;
        number : INT := 1;
        n2 : INT;
        n3 : INT := 4;
        n4 : INT;
        n5 : INT := 3;
        n6 : INT := 13;
        n7 : INT := 3;
        n8, n9, n10 : BOOL;
    END_VAR

    b2 := NOT FALSE;
    number := (- 19);
    n2 := (- 3)+ 2;
    b := NOT b;
    n5 := n5 * 2;
    n6 := n6 MOD 7;
    n7 := n7 - 4;
    n8 := 3 <> 4;
    n9 := 3 < 4 AND 3 <= 3 AND -4 < 5 AND 4 <= 7;
    n10 := 4 < 3 OR 4 <= 3 OR 6 < -5;
END_PROGRAM

CONFIGURATION Config0
  RESOURCE Res0 ON PLC
    TASK task0(INTERVAL := T#50ms, PRIORITY := 0);
    PROGRAM instance0 WITH task0 : my_sth;
  END_RESOURCE
END_CONFIGURATION

(* ---- runtimeTest.whileLoopTest.st ---- *)
PROGRAM MY_STH
    VAR_INPUT
        VAR1 : INT := 2;
        COUNTER : INT := 4;
    END_VAR

   WHILE COUNTER<>0 DO
       VAR1 := VAR1*2;
       COUNTER := COUNTER-1;
   END_WHILE;
END_PROGRAM

CONFIGURATION Config0
  RESOURCE Res0 ON PLC
    TASK TASK0(INTERVAL := T#50MS, PRIORITY := 0);
    PROGRAM INSTANCE0 WITH TASK0 : MY_STH;
  END_RESOURCE
END_CONFIGURATION

(* ---- Scenario0v0_Final.xml.st0.st ---- *)
TYPE
    MAGAZIN_STATES_T : (GREEN_LAMP , INIT , INTERSTEP , MAGAZIN_INIT , MAGAZIN_INIT_2 , SLIDER_MOVE_BACK , START_MAGAZIN , STEP0 , STEP1 , CONVEY);
    CRANE_STATES_T : (CRANE_INIT , CRANE_INIT_2 , CRANE_LIFT_CONVEYOR , CRANE_LIFT_MAGAZINE , CRANE_ON_CONVEYOR , CRANE_STOP , CRANE_TURN_LEFT , INIT , INTERSTEP , INTERSTEP_2 , INTERSTEP_CHECK_WORKPIECE , MAGAZIN_STOP , START_CRANE , TIMEDELAY , TURN_RIGHT , RELEASE);
END_TYPE

PROGRAM MAIN

VAR  ACTUATOR_CRANELOWER : BOOL; END_VAR
VAR  ACTUATOR_CRANETURNCLOCKWISE : BOOL; END_VAR
VAR  ACTUATOR_CRANETURNCOUNTERCLOCKWISE : BOOL; END_VAR
VAR  ACTUATOR_MAGAZINGREENLAMP : BOOL; END_VAR
VAR  ACTUATOR_MAGAZINSLIDER : BOOL; END_VAR
VAR  ACTUATOR_MAGAZINVACUUMOFF : BOOL; END_VAR
VAR  ACTUATOR_MAGAZINVACUUMON : BOOL; END_VAR
VAR  ACTUATOR_MAGAZINWHITELAMP : BOOL; END_VAR
VAR_INPUT  CRANE_CRANEDOWN : BOOL; END_VAR
VAR_OUTPUT  CRANE_CRANELOWER : BOOL; END_VAR
VAR_INPUT  CRANE_CRANEONCONVEYOR : BOOL; END_VAR
VAR_INPUT  CRANE_CRANEONMAGAZIN : BOOL; END_VAR
VAR_INPUT  CRANE_CRANESUCKED : BOOL; END_VAR
VAR_OUTPUT  CRANE_CRANETURNCLOCKWISE : BOOL; END_VAR
VAR_OUTPUT  CRANE_CRANETURNCOUNTERCLOCKWISE : BOOL; END_VAR
VAR_INPUT  CRANE_CRANEUP : BOOL; END_VAR
VAR_OUTPUT  CRANE_MAGAZINVACUUMOFF : BOOL; END_VAR
VAR_OUTPUT  CRANE_MAGAZINVACUUMON : BOOL; END_VAR
VAR  CRANE_SFCINIT : BOOL; END_VAR
VAR_INPUT  CRANE_SFCRESET : BOOL; END_VAR
VAR_INPUT  CRANE_SLIDERMOVEDOUT : BOOL; END_VAR
VAR_INPUT  CRANE_SLIDERNOTMOVEDOUT : BOOL; END_VAR
VAR_INPUT  CRANE_STARTBUTTONMAGAZIN : BOOL; END_VAR
VAR_OUTPUT  CRANE_STARTCOMMANDCRANE : BOOL; END_VAR
VAR_INPUT  CRANE_STARTVAR : BOOL; END_VAR
VAR_OUTPUT  CRANE_TIMEDELAY_TIMER_ET : UINT; END_VAR
VAR_INPUT  CRANE_TIMEDELAY_TIMER_IN : BOOL; END_VAR
VAR_INPUT  CRANE_TIMEDELAY_TIMER_PT : UINT; END_VAR
VAR_OUTPUT  CRANE_TIMEDELAY_TIMER_Q : BOOL; END_VAR
VAR  CRANE_TIMEDELAY_TIMER_DURATION : UINT := UINT#12; END_VAR
VAR  CRANE_TIMEDELAY_TIMER_INTERCONNECT : BOOL; END_VAR
VAR_INPUT  CRANE_WORKPIECEREADY : BOOL; END_VAR
VAR  CRANE_2STATE : CRANE_STATES_T; END_VAR
VAR  CRANE_2TRANSIT : BOOL; END_VAR
VAR  CRANE_INTERCONNECTCRANESTARTCOMMAND : BOOL; END_VAR
VAR_INPUT  MAG_CRANEDOWN : BOOL; END_VAR
VAR_INPUT  MAG_CRANEONCONVEYOR : BOOL; END_VAR
VAR_INPUT  MAG_CRANEONMAGAZIN : BOOL; END_VAR
VAR_INPUT  MAG_CRANESUCKED : BOOL; END_VAR
VAR_INPUT  MAG_CRANEUP : BOOL; END_VAR
VAR_OUTPUT  MAG_MAGAZINGREENLAMP : BOOL; END_VAR
VAR_OUTPUT  MAG_MAGAZINSLIDER : BOOL; END_VAR
VAR  MAG_SFCINIT : BOOL; END_VAR
VAR_INPUT  MAG_SFCRESET : BOOL; END_VAR
VAR_INPUT  MAG_SLIDERMOVEDOUT : BOOL; END_VAR
VAR_INPUT  MAG_SLIDERNOTMOVEDOUT : BOOL; END_VAR
VAR_INPUT  MAG_STARTBUTTONMAGAZIN : BOOL; END_VAR
VAR_OUTPUT  MAG_STARTCOMMANDMAGAZIN : BOOL; END_VAR
VAR_INPUT  MAG_STARTVAR : BOOL; END_VAR
VAR_INPUT  MAG_WORKPIECEREADY : BOOL; END_VAR
VAR  MAG_2STATE : MAGAZIN_STATES_T; END_VAR
VAR  MAG_2TRANSIT : BOOL; END_VAR
VAR  MAG_INTERCONNECTMAGAZINESTARTCOMMAND : BOOL; END_VAR
VAR  SENSOR_CRANEDOWN : BOOL; END_VAR
VAR  SENSOR_CRANEONCONVEYOR : BOOL; END_VAR
VAR  SENSOR_CRANEONMAGAZIN : BOOL; END_VAR
VAR  SENSOR_CRANEPOSITION : BOOL; END_VAR
VAR  SENSOR_CRANESUCKED : BOOL; END_VAR
VAR  SENSOR_CRANEUP : BOOL; END_VAR
VAR  SENSOR_MAGAZINEMERGENCYSTOP : BOOL; END_VAR
VAR  SENSOR_MAGAZINSWITCHMANUELLAUTOMATIC : BOOL; END_VAR
VAR  SENSOR_SLIDERMOVEDOUT : BOOL; END_VAR
VAR  SENSOR_SLIDERNOTMOVEDOUT : BOOL; END_VAR
VAR  SENSOR_STARTBUTTONMAGAZIN : BOOL; END_VAR
VAR  SENSOR_WORKPIECEREADY : BOOL; END_VAR
MAG_SLIDERNOTMOVEDOUT := SENSOR_SLIDERNOTMOVEDOUT;
MAG_SLIDERMOVEDOUT := SENSOR_SLIDERMOVEDOUT;
MAG_CRANEONMAGAZIN := SENSOR_CRANEONMAGAZIN;
MAG_CRANEDOWN := SENSOR_CRANEDOWN;
MAG_CRANEUP := SENSOR_CRANEUP;
MAG_CRANEONCONVEYOR := SENSOR_CRANEONCONVEYOR;
MAG_WORKPIECEREADY := SENSOR_WORKPIECEREADY;
MAG_STARTBUTTONMAGAZIN := SENSOR_STARTBUTTONMAGAZIN;
ACTUATOR_MAGAZINSLIDER := MAG_MAGAZINSLIDER;
ACTUATOR_MAGAZINGREENLAMP := MAG_MAGAZINGREENLAMP;
CRANE_WORKPIECEREADY := SENSOR_WORKPIECEREADY;
CRANE_CRANEUP := SENSOR_CRANEUP;
CRANE_CRANEONCONVEYOR := SENSOR_CRANEONCONVEYOR;
CRANE_CRANEDOWN := SENSOR_CRANEDOWN;
CRANE_CRANESUCKED := SENSOR_CRANESUCKED;
CRANE_CRANEONMAGAZIN := SENSOR_CRANEONMAGAZIN;
CRANE_SLIDERMOVEDOUT := SENSOR_SLIDERMOVEDOUT;
CRANE_STARTBUTTONMAGAZIN := SENSOR_STARTBUTTONMAGAZIN;
ACTUATOR_CRANETURNCOUNTERCLOCKWISE := CRANE_CRANETURNCOUNTERCLOCKWISE;
ACTUATOR_CRANETURNCLOCKWISE := CRANE_CRANETURNCLOCKWISE;
ACTUATOR_CRANELOWER := CRANE_CRANELOWER;
ACTUATOR_MAGAZINVACUUMOFF := CRANE_MAGAZINVACUUMOFF;
ACTUATOR_MAGAZINVACUUMON := CRANE_MAGAZINVACUUMON;
IF SENSOR_MAGAZINEMERGENCYSTOP THEN
    CASE MAG_2STATE OF
        MAGAZIN_STATES_T#GREEN_LAMP:
            MAG_2TRANSIT := FALSE;
            MAG_MAGAZINGREENLAMP := TRUE;
            MAG_INTERCONNECTMAGAZINESTARTCOMMAND := FALSE;
            IF TRUE THEN
                MAG_2TRANSIT := TRUE;
                MAG_2STATE := MAGAZIN_STATES_T#MAGAZIN_INIT;
            END_IF;

        MAGAZIN_STATES_T#INIT:
            MAG_2TRANSIT := FALSE;
            IF TRUE THEN
                MAG_2TRANSIT := TRUE;
                MAG_2STATE := MAGAZIN_STATES_T#START_MAGAZIN;
            END_IF;

        MAGAZIN_STATES_T#INTERSTEP:
            MAG_2TRANSIT := FALSE;
            MAG_STARTCOMMANDMAGAZIN := TRUE;
            IF MAG_STARTVAR THEN
                MAG_2TRANSIT := TRUE;
                MAG_2STATE := MAGAZIN_STATES_T#CONVEY;
            END_IF;

        MAGAZIN_STATES_T#MAGAZIN_INIT:
            MAG_2TRANSIT := FALSE;
            MAG_MAGAZINSLIDER := TRUE;
            IF TRUE THEN
                MAG_2TRANSIT := TRUE;
                MAG_2STATE := MAGAZIN_STATES_T#MAGAZIN_INIT_2;
            END_IF;

        MAGAZIN_STATES_T#MAGAZIN_INIT_2:
            MAG_2TRANSIT := FALSE;
            MAG_MAGAZINSLIDER := FALSE;
            IF TRUE THEN
                MAG_2TRANSIT := TRUE;
                MAG_2STATE := MAGAZIN_STATES_T#INTERSTEP;
            END_IF;

        MAGAZIN_STATES_T#SLIDER_MOVE_BACK:
            MAG_2TRANSIT := FALSE;
            IF ((MAG_SLIDERMOVEDOUT = TRUE) AND (MAG_SLIDERNOTMOVEDOUT = FALSE)) THEN
                MAG_MAGAZINSLIDER := FALSE;
            END_IF;
            IF MAG_CRANEUP THEN
                MAG_2TRANSIT := TRUE;
                MAG_2STATE := MAGAZIN_STATES_T#STEP1;
            END_IF;

        MAGAZIN_STATES_T#START_MAGAZIN:
            MAG_2TRANSIT := FALSE;
            MAG_MAGAZINSLIDER := FALSE;
            MAG_MAGAZINGREENLAMP := FALSE;
            MAG_STARTVAR := FALSE;
            MAG_STARTCOMMANDMAGAZIN := FALSE;
            IF (MAG_STARTBUTTONMAGAZIN = TRUE) THEN
                MAG_INTERCONNECTMAGAZINESTARTCOMMAND := TRUE;
            END_IF;
            IF MAG_INTERCONNECTMAGAZINESTARTCOMMAND THEN
                MAG_2TRANSIT := TRUE;
                MAG_2STATE := MAGAZIN_STATES_T#GREEN_LAMP;
            END_IF;

        MAGAZIN_STATES_T#STEP0:
            MAG_2TRANSIT := FALSE;
            IF MAG_CRANEDOWN THEN
                MAG_2TRANSIT := TRUE;
                MAG_2STATE := MAGAZIN_STATES_T#SLIDER_MOVE_BACK;
            END_IF;

        MAGAZIN_STATES_T#STEP1:
            MAG_2TRANSIT := FALSE;
            IF MAG_CRANEONCONVEYOR THEN
                MAG_2TRANSIT := TRUE;
                MAG_2STATE := MAGAZIN_STATES_T#INTERSTEP;
            END_IF;

        MAGAZIN_STATES_T#CONVEY:
            MAG_2TRANSIT := FALSE;
            IF MAG_SLIDERNOTMOVEDOUT THEN
                MAG_MAGAZINSLIDER := TRUE;
            END_IF;
            IF MAG_CRANEONMAGAZIN THEN
                MAG_2TRANSIT := TRUE;
                MAG_2STATE := MAGAZIN_STATES_T#STEP0;
            END_IF;

            END_CASE;
    CASE CRANE_2STATE OF
        CRANE_STATES_T#CRANE_INIT:
            CRANE_2TRANSIT := FALSE;
            CRANE_CRANELOWER := TRUE;
            CRANE_INTERCONNECTCRANESTARTCOMMAND := FALSE;
            IF CRANE_CRANEDOWN THEN
                CRANE_2TRANSIT := TRUE;
                CRANE_2STATE := CRANE_STATES_T#CRANE_INIT_2;
            END_IF;

        CRANE_STATES_T#CRANE_INIT_2:
            CRANE_2TRANSIT := FALSE;
            CRANE_CRANELOWER := FALSE;
            IF CRANE_CRANEUP THEN
                CRANE_2TRANSIT := TRUE;
                CRANE_2STATE := CRANE_STATES_T#INTERSTEP;
            END_IF;

        CRANE_STATES_T#CRANE_LIFT_CONVEYOR:
            CRANE_2TRANSIT := FALSE;
            CRANE_CRANELOWER := FALSE;
            IF TRUE THEN
                CRANE_2TRANSIT := TRUE;
                CRANE_2STATE := CRANE_STATES_T#INTERSTEP;
            END_IF;

        CRANE_STATES_T#CRANE_LIFT_MAGAZINE:
            CRANE_2TRANSIT := FALSE;
            CRANE_CRANELOWER := FALSE;
            IF CRANE_CRANEUP THEN
                CRANE_2TRANSIT := TRUE;
                CRANE_2STATE := CRANE_STATES_T#CRANE_TURN_LEFT;
            END_IF;

        CRANE_STATES_T#CRANE_ON_CONVEYOR:
            CRANE_2TRANSIT := FALSE;
            CRANE_CRANETURNCOUNTERCLOCKWISE := FALSE;
            CRANE_CRANETURNCLOCKWISE := FALSE;
            CRANE_CRANELOWER := TRUE;
            IF CRANE_CRANEDOWN THEN
                CRANE_2TRANSIT := TRUE;
                CRANE_2STATE := CRANE_STATES_T#RELEASE;
            END_IF;

        CRANE_STATES_T#CRANE_STOP:
            CRANE_2TRANSIT := FALSE;
            IF TRUE THEN
                CRANE_2TRANSIT := TRUE;
                CRANE_2STATE := CRANE_STATES_T#START_CRANE;
            END_IF;

        CRANE_STATES_T#CRANE_TURN_LEFT:
            CRANE_2TRANSIT := FALSE;
            CRANE_CRANETURNCOUNTERCLOCKWISE := TRUE;
            CRANE_CRANETURNCLOCKWISE := FALSE;
            IF CRANE_CRANEONCONVEYOR THEN
                CRANE_2TRANSIT := TRUE;
                CRANE_2STATE := CRANE_STATES_T#CRANE_ON_CONVEYOR;
            END_IF;

        CRANE_STATES_T#INIT:
            CRANE_2TRANSIT := FALSE;
            IF TRUE THEN
                CRANE_2TRANSIT := TRUE;
                CRANE_2STATE := CRANE_STATES_T#START_CRANE;
            END_IF;

        CRANE_STATES_T#INTERSTEP:
            CRANE_2TRANSIT := FALSE;
            CRANE_STARTCOMMANDCRANE := TRUE;
            IF CRANE_STARTVAR THEN
                CRANE_2TRANSIT := TRUE;
                CRANE_2STATE := CRANE_STATES_T#INTERSTEP_2;
            END_IF;

        CRANE_STATES_T#INTERSTEP_2:
            CRANE_2TRANSIT := FALSE;
            IF CRANE_SLIDERMOVEDOUT THEN
                CRANE_2TRANSIT := TRUE;
                CRANE_2STATE := CRANE_STATES_T#TIMEDELAY;
            END_IF;

        CRANE_STATES_T#INTERSTEP_CHECK_WORKPIECE:
            CRANE_2TRANSIT := FALSE;
            IF CRANE_WORKPIECEREADY THEN
                CRANE_2TRANSIT := TRUE;
                CRANE_2STATE := CRANE_STATES_T#MAGAZIN_STOP;
            ELSIF NOT CRANE_WORKPIECEREADY THEN
                CRANE_2TRANSIT := TRUE;
                CRANE_2STATE := CRANE_STATES_T#CRANE_STOP;
            END_IF;

        CRANE_STATES_T#MAGAZIN_STOP:
            CRANE_2TRANSIT := FALSE;
            CRANE_CRANETURNCLOCKWISE := FALSE;
            CRANE_CRANETURNCOUNTERCLOCKWISE := FALSE;
            CRANE_MAGAZINVACUUMON := TRUE;
            CRANE_MAGAZINVACUUMOFF := FALSE;
            CRANE_CRANELOWER := TRUE;
            IF CRANE_CRANESUCKED THEN
                CRANE_2TRANSIT := TRUE;
                CRANE_2STATE := CRANE_STATES_T#CRANE_LIFT_MAGAZINE;
            END_IF;

        CRANE_STATES_T#START_CRANE:
            CRANE_2TRANSIT := FALSE;
            CRANE_CRANELOWER := FALSE;
            CRANE_MAGAZINVACUUMOFF := TRUE;
            CRANE_MAGAZINVACUUMON := FALSE;
            CRANE_CRANETURNCOUNTERCLOCKWISE := FALSE;
            CRANE_CRANETURNCLOCKWISE := FALSE;
            CRANE_STARTVAR := FALSE;
            CRANE_STARTCOMMANDCRANE := FALSE;
            IF (CRANE_STARTBUTTONMAGAZIN = TRUE) THEN
                CRANE_INTERCONNECTCRANESTARTCOMMAND := TRUE;
            END_IF;
            IF CRANE_INTERCONNECTCRANESTARTCOMMAND THEN
                CRANE_2TRANSIT := TRUE;
                CRANE_2STATE := CRANE_STATES_T#CRANE_INIT;
            END_IF;

        CRANE_STATES_T#TIMEDELAY:
            CRANE_2TRANSIT := FALSE;
            CRANE_TIMEDELAY_TIMER_IN := TRUE;
            CRANE_TIMEDELAY_TIMER_PT := CRANE_TIMEDELAY_TIMER_DURATION;
            IF CRANE_TIMEDELAY_TIMER_IN THEN
                CRANE_TIMEDELAY_TIMER_Q := (CRANE_TIMEDELAY_TIMER_ET = UINT#0);
                IF (CRANE_TIMEDELAY_TIMER_ET > UINT#0) THEN
                    CRANE_TIMEDELAY_TIMER_ET := (CRANE_TIMEDELAY_TIMER_ET - UINT#1);
                ELSE
                    CRANE_TIMEDELAY_TIMER_ET := UINT#0;
                END_IF;
            ELSE
                CRANE_TIMEDELAY_TIMER_Q := FALSE;
                CRANE_TIMEDELAY_TIMER_ET := CRANE_TIMEDELAY_TIMER_PT;
            END_IF;
            CRANE_TIMEDELAY_TIMER_INTERCONNECT := CRANE_TIMEDELAY_TIMER_Q;
            IF CRANE_TIMEDELAY_TIMER_INTERCONNECT THEN
                CRANE_2TRANSIT := TRUE;
                CRANE_2STATE := CRANE_STATES_T#TURN_RIGHT;
            END_IF;

        CRANE_STATES_T#TURN_RIGHT:
            CRANE_2TRANSIT := FALSE;
            CRANE_CRANETURNCLOCKWISE := TRUE;
            CRANE_CRANETURNCOUNTERCLOCKWISE := FALSE;
            IF CRANE_CRANEONMAGAZIN THEN
                CRANE_2TRANSIT := TRUE;
                CRANE_2STATE := CRANE_STATES_T#INTERSTEP_CHECK_WORKPIECE;
            END_IF;

        CRANE_STATES_T#RELEASE:
            CRANE_2TRANSIT := FALSE;
            CRANE_MAGAZINVACUUMOFF := TRUE;
            CRANE_MAGAZINVACUUMON := FALSE;
            IF TRUE THEN
                CRANE_2TRANSIT := TRUE;
                CRANE_2STATE := CRANE_STATES_T#CRANE_LIFT_CONVEYOR;
            END_IF;

            END_CASE;
    IF ACTUATOR_MAGAZINGREENLAMP THEN
        IF (CRANE_STARTCOMMANDCRANE AND MAG_STARTCOMMANDMAGAZIN) THEN
            CRANE_STARTVAR := TRUE;
            MAG_STARTVAR := TRUE;
        END_IF;
    END_IF;
    CRANE_SFCRESET := FALSE;
    MAG_SFCRESET := FALSE;
ELSIF NOT SENSOR_MAGAZINEMERGENCYSTOP THEN
    ACTUATOR_MAGAZINSLIDER := FALSE;
    ACTUATOR_CRANELOWER := FALSE;
    ACTUATOR_MAGAZINVACUUMON := FALSE;
    ACTUATOR_MAGAZINVACUUMOFF := TRUE;
    ACTUATOR_MAGAZINGREENLAMP := FALSE;
    ACTUATOR_CRANETURNCOUNTERCLOCKWISE := FALSE;
    ACTUATOR_CRANETURNCLOCKWISE := FALSE;
    CRANE_2STATE := CRANE_STATES_T#INIT;
    MAG_2STATE := MAGAZIN_STATES_T#INIT;
    CRANE_STARTVAR := FALSE;
    MAG_STARTVAR := FALSE;
END_IF;
END_PROGRAM

CONFIGURATION Config0
  RESOURCE Res0 ON PLC
    TASK TASK0(INTERVAL := T#50MS, PRIORITY := 0);
    PROGRAM INSTANCE0 WITH TASK0 : MAIN;
  END_RESOURCE
END_CONFIGURATION
